KUKA KRL program: MyProgram_218().src

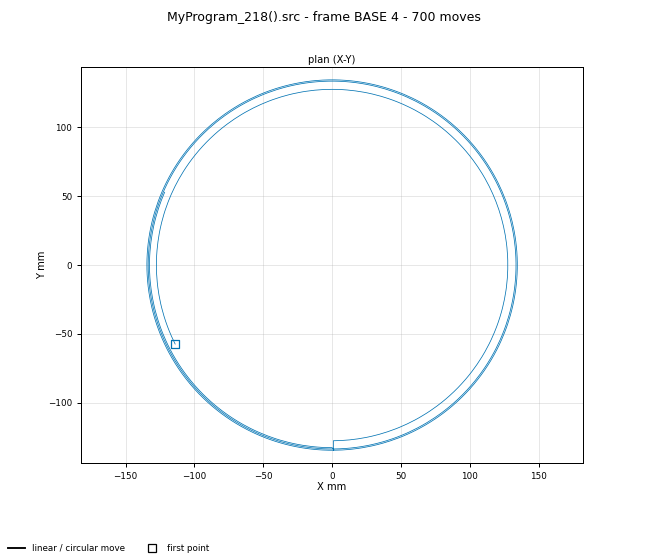
[picture p0: tool path of MyProgram_218().src in frame BASE 4, 700 of 700 moves have a stored position in this frame; points joined in program order, loops and branches not executed]
&ACCESS RVP
&REL 1
&PARAM TEMPLATE = C:\KRC\Roboter\Template\vorgabe
&PARAM EDITMASK = *
DEF MyProgram_218()
; ---- Setting reference (Base) ----
$BASE = BASE_DATA[4]

; --------------------------
; ---- Setting tool (TCP) ----
$TOOL = TOOL_DATA[3]
; --------------------------

$VEL.CP = VEL_APROX_PRINT
Startdeposition()
$VEL.CP = VEL_PRINT
LIN {X -113.9727,Y -57.3713,Z 152,A -154.6859,B 17.5235,C -0.3256,E1 17.383,E2 243.3579} C_DIS
LIN {X -115.3507,Y -54.5472,Z 152,A -156.1373,B 17.5235,C -0.3282,E1 17.3813,E2 244.8124} C_DIS
LIN {X -116.579,Y -51.8684,Z 152,A -157.511,B 17.5234,C -0.3302,E1 17.3797,E2 246.1904} C_DIS
LIN {X -118.2068,Y -48.044,Z 152,A -159.4681,B 17.5234,C -0.3326,E1 17.3776,E2 248.1558} C_DIS
LIN {X -119.5357,Y -44.6339,Z 152,A -161.0343,B 17.5232,C -0.3396,E1 17.376,E2 249.7114} C_DIS
LIN {X -120.8839,Y -40.8453,Z 152,A -162.9985,B 17.5232,C -0.3398,E1 17.3742,E2 251.6915} C_DIS
LIN {X -122.0836,Y -37.1027,Z 152,A -164.6161,B 17.523,C -0.3495,E1 17.3729,E2 253.2904} C_DIS
LIN {X -122.9269,Y -34.2049,Z 152,A -165.9736,B 17.523,C -0.3534,E1 17.3718,E2 254.6466} C_DIS
LIN {X -123.7291,Y -31.1788,Z 152,A -167.3908,B 17.5229,C -0.3571,E1 17.3708,E2 256.0634} C_DIS
LIN {X -124.4565,Y -28.1362,Z 152,A -168.7811,B 17.5228,C -0.3617,E1 17.37,E2 257.4504} C_DIS
LIN {X -125.1457,Y -24.8967,Z 152,A -170.2929,B 17.5227,C -0.3654,E1 17.3691,E2 258.9631} C_DIS
LIN {X -125.7207,Y -21.8119,Z 152,A -171.7167,B 17.5227,C -0.3691,E1 17.3684,E2 260.3869} C_DIS
LIN {X -126.2175,Y -18.7245,Z 152,A -173.1623,B 17.5226,C -0.3721,E1 17.3678,E2 261.8354} C_DIS
LIN {X -126.5469,Y -16.3393,Z 152,A -174.3275,B 17.5226,C -0.3728,E1 17.3674,E2 263.0086} C_DIS
LIN {X -126.9668,Y -12.6766,Z 152,A -175.922,B 17.5224,C -0.3797,E1 17.3669,E2 264.5941} C_DIS
LIN {X -127.2461,Y -9.4608,Z 152,A -177.3928,B 17.5224,C -0.3834,E1 17.3666,E2 266.0654} C_DIS
LIN {X -127.4345,Y -6.4427,Z 152,A -178.7722,B 17.5222,C -0.3869,E1 17.3663,E2 267.4454} C_DIS
LIN {X -127.5543,Y -3.3188,Z 152,A 179.8307,B 17.5222,C -0.3914,E1 17.3663,E2 268.8398} C_DIS
LIN {X -127.6001,Y -0.0843,Z 152,A 178.3637,B 17.5221,C -0.3954,E1 17.3662,E2 270.3066} C_DIS
LIN {X -127.5647,Y 2.9425,Z 152,A 176.9278,B 17.5221,C -0.3972,E1 17.3662,E2 271.7492} C_DIS
LIN {X -127.4125,Y 6.8803,Z 152,A 175.04,B 17.522,C -0.399,E1 17.3665,E2 273.6477} C_DIS
LIN {X -127.1428,Y 10.7584,Z 152,A 173.4238,B 17.5218,C -0.4084,E1 17.3668,E2 275.247} C_DIS
LIN {X -126.8198,Y 14.0691,Z 152,A 171.9562,B 17.5217,C -0.4138,E1 17.3673,E2 276.7095} C_DIS
LIN {X -126.4609,Y 16.9953,Z 152,A 170.6184,B 17.5216,C -0.4174,E1 17.3677,E2 278.0471} C_DIS
LIN {X -126.007,Y 20.0892,Z 152,A 169.1704,B 17.5216,C -0.4203,E1 17.3684,E2 279.498} C_DIS
LIN {X -125.4777,Y 23.1701,Z 152,A 167.7181,B 17.5214,C -0.4231,E1 17.3691,E2 280.9538} C_DIS
LIN {X -124.7928,Y 26.6056,Z 152,A 166.0587,B 17.5214,C -0.4252,E1 17.37,E2 282.6206} C_DIS
LIN {X -123.7662,Y 31.0327,Z 152,A 164.1264,B 17.5212,C -0.4347,E1 17.3713,E2 284.5378} C_DIS
LIN {X -122.9699,Y 34.0512,Z 152,A 162.8468,B 17.521,C -0.4427,E1 17.3722,E2 285.8017} C_DIS
LIN {X -122.1521,Y 36.8791,Z 152,A 161.3808,B 17.521,C -0.4422,E1 17.3733,E2 287.2819} C_DIS
LIN {X -121.2101,Y 39.8659,Z 152,A 159.9672,B 17.5209,C -0.4461,E1 17.3745,E2 288.6944} C_DIS
LIN {X -120.1418,Y 42.9767,Z 152,A 158.4732,B 17.5208,C -0.4499,E1 17.3759,E2 290.1881} C_DIS
LIN {X -119.0471,Y 45.9221,Z 152,A 157.0498,B 17.5207,C -0.4537,E1 17.3773,E2 291.6109} C_DIS
LIN {X -118.0113,Y 48.5257,Z 152,A 155.7284,B 17.5207,C -0.4553,E1 17.3787,E2 292.9376} C_DIS
LIN {X -116.8398,Y 51.2823,Z 152,A 154.2995,B 17.5207,C -0.4566,E1 17.3803,E2 294.3739} C_DIS
LIN {X -115.4259,Y 54.3898,Z 152,A 152.885,B 17.5204,C -0.4646,E1 17.382,E2 295.773} C_DIS
LIN {X -114.0589,Y 57.202,Z 152,A 151.456,B 17.5204,C -0.4678,E1 17.3837,E2 297.2028} C_DIS
LIN {X -112.5261,Y 60.1611,Z 152,A 149.9928,B 17.5202,C -0.473,E1 17.3856,E2 298.6602} C_DIS
LIN {X -111.11,Y 62.7379,Z 152,A 148.593,B 17.5202,C -0.4741,E1 17.3875,E2 300.0669} C_DIS
LIN {X -109.5435,Y 65.4343,Z 152,A 147.208,B 17.5201,C -0.4784,E1 17.3895,E2 301.4483} C_DIS
LIN {X -107.9124,Y 68.0906,Z 152,A 145.7625,B 17.52,C -0.4807,E1 17.3916,E2 302.8969} C_DIS
LIN {X -106.0955,Y 70.8884,Z 152,A 144.2532,B 17.52,C -0.4843,E1 17.3939,E2 304.4053} C_DIS
LIN {X -103.8442,Y 74.1471,Z 152,A 142.3482,B 17.5199,C -0.485,E1 17.397,E2 306.322} C_DIS
LIN {X -101.547,Y 77.264,Z 152,A 140.7503,B 17.5196,C -0.4938,E1 17.3997,E2 307.9018} C_DIS
LIN {X -99.1877,Y 80.2699,Z 152,A 139.0108,B 17.5196,C -0.4973,E1 17.4027,E2 309.6417} C_DIS
LIN {X -96.9265,Y 82.9868,Z 152,A 137.3158,B 17.5196,C -0.4978,E1 17.4058,E2 311.3465} C_DIS
LIN {X -94.0753,Y 86.2049,Z 152,A 135.4528,B 17.5193,C -0.5045,E1 17.4092,E2 313.1994} C_DIS
LIN {X -91.3904,Y 89.047,Z 152,A 133.6596,B 17.5193,C -0.5073,E1 17.4127,E2 314.9945} C_DIS
LIN {X -88.5541,Y 91.8676,Z 152,A 131.745,B 17.5193,C -0.5076,E1 17.4165,E2 316.9199} C_DIS
LIN {X -85.3855,Y 94.82,Z 152,A 129.8494,B 17.5191,C -0.5134,E1 17.4204,E2 318.8076} C_DIS
LIN {X -82.6808,Y 97.1869,Z 152,A 128.179,B 17.5191,C -0.515,E1 17.4239,E2 320.4823} C_DIS
LIN {X -79.7356,Y 99.6181,Z 152,A 126.4292,B 17.519,C -0.5174,E1 17.4277,E2 322.2338} C_DIS
LIN {X -76.1604,Y 102.3768,Z 152,A 124.5451,B 17.5187,C -0.5259,E1 17.4319,E2 324.0995} C_DIS
LIN {X -73.4698,Y 104.3245,Z 152,A 123.0566,B 17.5187,C -0.5288,E1 17.4353,E2 325.586} C_DIS
LIN {X -70.9621,Y 106.0463,Z 152,A 121.6854,B 17.5186,C -0.5311,E1 17.4384,E2 326.9561} C_DIS
LIN {X -68.3819,Y 107.7285,Z 152,A 120.2468,B 17.5186,C -0.5318,E1 17.4418,E2 328.3994} C_DIS
LIN {X -66.0845,Y 109.1524,Z 152,A 118.9664,B 17.5186,C -0.5318,E1 17.4449,E2 329.6858} C_DIS
LIN {X -63.0785,Y 110.9168,Z 152,A 117.4551,B 17.5184,C -0.536,E1 17.4485,E2 331.1894} C_DIS
LIN {X -60.1402,Y 112.5374,Z 152,A 115.9589,B 17.5184,C -0.5387,E1 17.4522,E2 332.6828} C_DIS
LIN {X -57.3655,Y 113.9757,Z 152,A 114.5616,B 17.5183,C -0.541,E1 17.4557,E2 334.0779} C_DIS
LIN {X -54.5551,Y 115.3469,Z 152,A 113.1534,B 17.5183,C -0.5429,E1 17.4592,E2 335.4852} C_DIS
LIN {X -51.8611,Y 116.5822,Z 152,A 111.7973,B 17.5183,C -0.544,E1 17.4627,E2 336.8427} C_DIS
LIN {X -48.8285,Y 117.8849,Z 152,A 110.3545,B 17.5181,C -0.5472,E1 17.4664,E2 338.2797} C_DIS
LIN {X -46.0972,Y 118.979,Z 152,A 109.0078,B 17.5181,C -0.548,E1 17.4699,E2 339.628} C_DIS
LIN {X -43.1738,Y 120.0707,Z 152,A 107.6953,B 17.5179,C -0.5525,E1 17.4733,E2 340.9292} C_DIS
LIN {X -40.016,Y 121.1601,Z 152,A 106.1214,B 17.5179,C -0.5517,E1 17.4774,E2 342.5101} C_DIS
LIN {X -37.0357,Y 122.1041,Z 152,A 104.6891,B 17.5179,C -0.5523,E1 17.4813,E2 343.9443} C_DIS
LIN {X -34.2041,Y 122.9271,Z 152,A 103.3614,B 17.5179,C -0.5534,E1 17.4848,E2 345.2714} C_DIS
LIN {X -31.1786,Y 123.7292,Z 152,A 101.9534,B 17.5179,C -0.5546,E1 17.4886,E2 346.6785} C_DIS
LIN {X -28.1119,Y 124.462,Z 152,A 100.5355,B 17.5179,C -0.5556,E1 17.4925,E2 348.0956} C_DIS
LIN {X -24.8793,Y 125.1493,Z 152,A 99.0624,B 17.5179,C -0.5571,E1 17.4965,E2 349.5664} C_DIS
LIN {X -21.8085,Y 125.7213,Z 152,A 97.6548,B 17.5178,C -0.5578,E1 17.5004,E2 350.9735} C_DIS
LIN {X -19.1709,Y 126.1492,Z 152,A 96.324,B 17.5178,C -0.5542,E1 17.5041,E2 352.3181} C_DIS
LIN {X -15.5304,Y 126.6491,Z 152,A 94.8319,B 17.5178,C -0.5603,E1 17.5082,E2 353.7915} C_DIS
LIN {X -12.6253,Y 126.9717,Z 152,A 93.4661,B 17.5178,C -0.5591,E1 17.512,E2 355.1625} C_DIS
LIN {X -9.3696,Y 127.2527,Z 152,A 92.0232,B 17.5178,C -0.5605,E1 17.516,E2 356.6018} C_DIS
LIN {X -6.6201,Y 127.4255,Z 152,A 90.6884,B 17.5178,C -0.5576,E1 17.5197,E2 357.9468} C_DIS
LIN {X -3.2848,Y 127.5552,Z 152,A 89.2597,B 17.5178,C -0.5603,E1 17.5237,E2 359.3668} C_DIS
LIN {X -0.2372,Y 127.5979,Z 152,A 87.8455,B 17.5178,C -0.5589,E1 17.5277,E2 360.7856} C_DIS
LIN {X 3.1496,Y 127.559,Z 152,A 86.198,B 17.5178,C -0.5547,E1 17.5323,E2 362.4465} C_DIS
LIN {X 7.5474,Y 127.3741,Z 152,A 84.3585,B 17.5178,C -0.5593,E1 17.5374,E2 364.2698} C_DIS
LIN {X 10.7934,Y 127.1398,Z 152,A 82.9113,B 17.5178,C -0.5596,E1 17.5414,E2 365.7148} C_DIS
LIN {X 14.0805,Y 126.8186,Z 152,A 81.4639,B 17.5177,C -0.5605,E1 17.5454,E2 367.1578} C_DIS
LIN {X 17.0025,Y 126.4599,Z 152,A 80.1413,B 17.5177,C -0.5602,E1 17.5491,E2 368.4801} C_DIS
LIN {X 20.0911,Y 126.0067,Z 152,A 78.7462,B 17.5177,C -0.5599,E1 17.5529,E2 369.8741} C_DIS
LIN {X 23.1858,Y 125.4748,Z 152,A 77.2629,B 17.5178,C -0.5568,E1 17.557,E2 371.3652} C_DIS
LIN {X 26.1682,Y 124.887,Z 152,A 75.8682,B 17.5178,C -0.5551,E1 17.5609,E2 372.7631} C_DIS
LIN {X 29.3622,Y 124.1739,Z 152,A 74.4493,B 17.5178,C -0.556,E1 17.5647,E2 374.176} C_DIS
LIN {X 32.5203,Y 123.3837,Z 152,A 73.0323,B 17.5178,C -0.5566,E1 17.5685,E2 375.5877} C_DIS
LIN {X 35.5353,Y 122.5492,Z 152,A 71.7806,B 17.5177,C -0.5609,E1 17.5718,E2 376.822} C_DIS
LIN {X 38.3685,Y 121.6924,Z 152,A 70.3268,B 17.5179,C -0.5555,E1 17.5758,E2 378.2899} C_DIS
LIN {X 40.7446,Y 120.9175,Z 152,A 69.0061,B 17.5181,C -0.5476,E1 17.5793,E2 379.6329} C_DIS
LIN {X 44.4806,Y 119.5931,Z 152,A 67.4143,B 17.5179,C -0.5526,E1 17.5834,E2 381.2035} C_DIS
LIN {X 47.5572,Y 118.403,Z 152,A 65.8169,B 17.5181,C -0.547,E1 17.5876,E2 382.814} C_DIS
LIN {X 51.5368,Y 116.7273,Z 152,A 63.9492,B 17.5181,C -0.5473,E1 17.5924,E2 384.674} C_DIS
LIN {X 54.395,Y 115.4234,Z 152,A 62.6043,B 17.5181,C -0.548,E1 17.5958,E2 386.0116} C_DIS
LIN {X 56.6861,Y 114.3139,Z 152,A 61.3941,B 17.5181,C -0.5442,E1 17.5988,E2 387.2295} C_DIS
LIN {X 60.1523,Y 112.5309,Z 152,A 59.7483,B 17.5181,C -0.5456,E1 17.6029,E2 388.8639} C_DIS
LIN {X 62.7654,Y 111.0945,Z 152,A 58.3557,B 17.5183,C -0.5418,E1 17.6063,E2 390.263} C_DIS
LIN {X 65.229,Y 109.6659,Z 152,A 57.0551,B 17.5183,C -0.5392,E1 17.6094,E2 391.5664} C_DIS
LIN {X 68.0911,Y 107.9121,Z 152,A 55.569,B 17.5183,C -0.5377,E1 17.6129,E2 393.0505} C_DIS
LIN {X 70.8752,Y 106.1043,Z 152,A 54.1195,B 17.5184,C -0.5368,E1 17.6163,E2 394.4959} C_DIS
LIN {X 73.4692,Y 104.3249,Z 152,A 52.6793,B 17.5185,C -0.5335,E1 17.6196,E2 395.9398} C_DIS
LIN {X 76.6358,Y 102.0218,Z 152,A 50.8146,B 17.5187,C -0.5266,E1 17.6238,E2 397.8173} C_DIS
LIN {X 80.2759,Y 99.1829,Z 152,A 48.9031,B 17.5187,C -0.5287,E1 17.628,E2 399.7115} C_DIS
LIN {X 82.8559,Y 97.038,Z 152,A 47.2561,B 17.5189,C -0.5208,E1 17.6315,E2 401.3752} C_DIS
LIN {X 86.2638,Y 94.0212,Z 152,A 45.2244,B 17.5189,C -0.5172,E1 17.6358,E2 403.4065} C_DIS
LIN {X 89.5956,Y 90.8524,Z 152,A 43.4329,B 17.5189,C -0.5229,E1 17.6393,E2 405.1683} C_DIS
LIN {X 91.8787,Y 88.5426,Z 152,A 41.7138,B 17.5192,C -0.5103,E1 17.6427,E2 406.918} C_DIS
LIN {X 95.0101,Y 85.1734,Z 152,A 39.8051,B 17.5192,C -0.5115,E1 17.6463,E2 408.8103} C_DIS
LIN {X 97.1851,Y 82.6829,Z 152,A 38.2159,B 17.5194,C -0.5044,E1 17.6492,E2 410.4124} C_DIS
LIN {X 99.6158,Y 79.7385,Z 152,A 36.4998,B 17.5194,C -0.5004,E1 17.6522,E2 412.13} C_DIS
LIN {X 102.2461,Y 76.3359,Z 152,A 34.81,B 17.5194,C -0.5047,E1 17.655,E2 413.7938} C_DIS
LIN {X 104.2367,Y 73.5943,Z 152,A 33.2206,B 17.5195,C -0.4985,E1 17.6576,E2 415.3923} C_DIS
LIN {X 105.7394,Y 71.4185,Z 152,A 31.9523,B 17.5197,C -0.4926,E1 17.6596,E2 416.6707} C_DIS
LIN {X 107.7055,Y 68.4184,Z 152,A 30.3969,B 17.5197,C -0.4906,E1 17.662,E2 418.2213} C_DIS
LIN {X 109.1695,Y 66.0563,Z 152,A 29.1069,B 17.5199,C -0.4858,E1 17.6639,E2 419.5172} C_DIS
LIN {X 110.9329,Y 63.0503,Z 152,A 27.6196,B 17.5199,C -0.4846,E1 17.6659,E2 420.9971} C_DIS
LIN {X 112.5301,Y 60.1537,Z 152,A 26.1549,B 17.5199,C -0.4815,E1 17.6679,E2 422.4609} C_DIS
LIN {X 113.974,Y 57.3689,Z 152,A 24.7695,B 17.5201,C -0.4786,E1 17.6697,E2 423.845} C_DIS
LIN {X 115.3525,Y 54.5434,Z 152,A 23.4063,B 17.5201,C -0.4765,E1 17.6713,E2 425.2042} C_DIS
LIN {X 116.5781,Y 51.8704,Z 152,A 22.0428,B 17.5202,C -0.4713,E1 17.6729,E2 426.574} C_DIS
LIN {X 117.8808,Y 48.8383,Z 152,A 20.6189,B 17.5202,C -0.4694,E1 17.6744,E2 427.9928} C_DIS
LIN {X 118.9736,Y 46.111,Z 152,A 19.2844,B 17.5204,C -0.4651,E1 17.6758,E2 429.3304} C_DIS
LIN {X 120.0763,Y 43.1585,Z 152,A 17.8852,B 17.5204,C -0.4617,E1 17.6771,E2 430.7294} C_DIS
LIN {X 121.0836,Y 40.2459,Z 152,A 16.5038,B 17.5206,C -0.4578,E1 17.6784,E2 432.112} C_DIS
LIN {X 122.1039,Y 37.0365,Z 152,A 15.0152,B 17.5206,C -0.4543,E1 17.6796,E2 433.5998} C_DIS
LIN {X 122.9263,Y 34.2069,Z 152,A 13.7032,B 17.5208,C -0.4509,E1 17.6806,E2 434.9119} C_DIS
LIN {X 123.728,Y 31.1835,Z 152,A 12.3118,B 17.5208,C -0.4472,E1 17.6816,E2 436.3035} C_DIS
LIN {X 124.4575,Y 28.1319,Z 152,A 10.917,B 17.5209,C -0.4436,E1 17.6825,E2 437.6985} C_DIS
LIN {X 125.1485,Y 24.883,Z 152,A 9.4528,B 17.521,C -0.4401,E1 17.6833,E2 439.1614} C_DIS
LIN {X 125.7205,Y 21.8133,Z 152,A 8.0609,B 17.5211,C -0.4363,E1 17.684,E2 440.5539} C_DIS
LIN {X 126.2166,Y 18.7312,Z 152,A 6.6205,B 17.5213,C -0.4306,E1 17.6846,E2 442.0005} C_DIS
LIN {X 126.6434,Y 15.5787,Z 152,A 5.2902,B 17.5213,C -0.43,E1 17.6851,E2 443.3214} C_DIS
LIN {X 126.9682,Y 12.6619,Z 152,A 3.9262,B 17.5214,C -0.4243,E1 17.6855,E2 444.6924} C_DIS
LIN {X 127.2517,Y 9.3841,Z 152,A 2.4704,B 17.5214,C -0.4206,E1 17.6858,E2 446.1476} C_DIS
LIN {X 127.4339,Y 6.4536,Z 152,A 1.1297,B 17.5216,C -0.4157,E1 17.686,E2 447.4926} C_DIS
LIN {X 127.5549,Y 3.2971,Z 152,A -0.2217,B 17.5216,C -0.4139,E1 17.6861,E2 448.8383} C_DIS
LIN {X 127.5999,Y -0.1226,Z 152,A -1.735,B 17.5217,C -0.4099,E1 17.6861,E2 450.3511} C_DIS
LIN {X 127.5635,Y -2.9879,Z 152,A -3.0967,B 17.5219,C -0.4032,E1 17.6861,E2 451.7232} C_DIS
LIN {X 127.4535,Y -6.0634,Z 152,A -4.4675,B 17.5219,C -0.3994,E1 17.6859,E2 453.0946} C_DIS
LIN {X 127.2627,Y -9.2329,Z 152,A -5.8219,B 17.522,C -0.3977,E1 17.6857,E2 454.4427} C_DIS
LIN {X 126.9816,Y -12.5221,Z 152,A -7.281,B 17.522,C -0.394,E1 17.6853,E2 455.9013} C_DIS
LIN {X 126.6378,Y -15.6255,Z 152,A -8.6566,B 17.5222,C -0.3906,E1 17.6849,E2 457.2758} C_DIS
LIN {X 126.2438,Y -18.5407,Z 152,A -9.9788,B 17.5222,C -0.3866,E1 17.6844,E2 458.6} C_DIS
LIN {X 125.7181,Y -21.8264,Z 152,A -11.4215,B 17.5223,C -0.3839,E1 17.6837,E2 460.0389} C_DIS
LIN {X 125.1456,Y -24.8975,Z 152,A -12.8014,B 17.5223,C -0.3805,E1 17.683,E2 461.4182} C_DIS
LIN {X 124.497,Y -27.9587,Z 152,A -14.126,B 17.5224,C -0.3793,E1 17.6822,E2 462.7355} C_DIS
LIN {X 123.7741,Y -31.0017,Z 152,A -15.647,B 17.5226,C -0.3706,E1 17.6812,E2 464.2721} C_DIS
LIN {X 122.9768,Y -34.0263,Z 152,A -17.0374,B 17.5226,C -0.3669,E1 17.6802,E2 465.6628} C_DIS
LIN {X 121.9537,Y -37.5271,Z 152,A -18.6757,B 17.5228,C -0.362,E1 17.6789,E2 467.3036} C_DIS
LIN {X 120.7154,Y -41.3398,Z 152,A -20.5043,B 17.5228,C -0.3556,E1 17.6773,E2 469.1381} C_DIS
LIN {X 119.5324,Y -44.6426,Z 152,A -22.1216,B 17.523,C -0.3494,E1 17.6757,E2 470.7624} C_DIS
LIN {X 117.8814,Y -48.8368,Z 152,A -23.9488,B 17.523,C -0.3509,E1 17.6738,E2 472.5699} C_DIS
LIN {X 116.7231,Y -51.5461,Z 152,A -25.3771,B 17.5231,C -0.3431,E1 17.6722,E2 474.0123} C_DIS
LIN {X 115.4269,Y -54.3877,Z 152,A -26.7063,B 17.5231,C -0.3418,E1 17.6707,E2 475.335} C_DIS
LIN {X 114.0623,Y -57.1954,Z 152,A -28.1026,B 17.5232,C -0.3381,E1 17.6689,E2 476.7327} C_DIS
LIN {X 112.5434,Y -60.1289,Z 152,A -29.5443,B 17.5232,C -0.3355,E1 17.6671,E2 478.1718} C_DIS
LIN {X 111.0232,Y -62.8921,Z 152,A -31.1308,B 17.5235,C -0.3252,E1 17.6649,E2 479.7801} C_DIS
LIN {X 108.7235,Y -66.7878,Z 152,A -32.9962,B 17.5235,C -0.3259,E1 17.6622,E2 481.6291} C_DIS
LIN {X 106.9561,Y -69.5831,Z 152,A -34.4704,B 17.5235,C -0.3223,E1 17.66,E2 483.1041} C_DIS
LIN {X 105.2184,Y -72.1837,Z 152,A -35.8035,B 17.5235,C -0.3213,E1 17.6579,E2 484.4309} C_DIS
LIN {X 103.4052,Y -74.7583,Z 152,A -37.2614,B 17.5236,C -0.3159,E1 17.6555,E2 485.8959} C_DIS
LIN {X 101.5429,Y -77.2693,Z 152,A -38.6513,B 17.5236,C -0.3129,E1 17.6532,E2 487.2861} C_DIS
LIN {X 99.1856,Y -80.2724,Z 152,A -40.3639,B 17.5238,C -0.3086,E1 17.6502,E2 489.001} C_DIS
LIN {X 97.0943,Y -82.7898,Z 152,A -41.9717,B 17.5238,C -0.2999,E1 17.6473,E2 490.6267} C_DIS
LIN {X 94.0701,Y -86.2105,Z 152,A -43.8726,B 17.5238,C -0.3005,E1 17.6438,E2 492.5131} C_DIS
LIN {X 91.3874,Y -89.0501,Z 152,A -45.6394,B 17.524,C -0.2959,E1 17.6404,E2 494.2838} C_DIS
LIN {X 88.5537,Y -91.868,Z 152,A -47.5442,B 17.524,C -0.2878,E1 17.6365,E2 496.2036} C_DIS
LIN {X 85.1685,Y -95.0144,Z 152,A -49.459,B 17.524,C -0.2891,E1 17.6326,E2 498.1025} C_DIS
LIN {X 82.6786,Y -97.1888,Z 152,A -51.0484,B 17.5242,C -0.2821,E1 17.6292,E2 499.706} C_DIS
LIN {X 79.7344,Y -99.6191,Z 152,A -52.7656,B 17.5242,C -0.2784,E1 17.6255,E2 501.4257} C_DIS
LIN {X 76.1486,Y -102.3856,Z 152,A -54.6422,B 17.5242,C -0.2801,E1 17.6214,E2 503.2866} C_DIS
LIN {X 73.6188,Y -104.2195,Z 152,A -56.0343,B 17.5242,C -0.2778,E1 17.6182,E2 504.6791} C_DIS
LIN {X 71.0407,Y -105.9938,Z 152,A -57.4285,B 17.5242,C -0.2756,E1 17.615,E2 506.0736} C_DIS
LIN {X 68.4247,Y -107.7015,Z 152,A -58.8742,B 17.5243,C -0.2715,E1 17.6116,E2 507.5259} C_DIS
LIN {X 65.6278,Y -109.4282,Z 152,A -60.3035,B 17.5243,C -0.2706,E1 17.6082,E2 508.9514} C_DIS
LIN {X 63.4871,Y -110.6837,Z 152,A -61.5477,B 17.5245,C -0.264,E1 17.6051,E2 510.212} C_DIS
LIN {X 60.1265,Y -112.5447,Z 152,A -63.1414,B 17.5245,C -0.266,E1 17.6013,E2 511.7923} C_DIS
LIN {X 57.3554,Y -113.9808,Z 152,A -64.5249,B 17.5245,C -0.2645,E1 17.5978,E2 513.1752} C_DIS
LIN {X 54.5498,Y -115.3494,Z 152,A -65.9184,B 17.5245,C -0.2627,E1 17.5943,E2 514.5692} C_DIS
LIN {X 51.8741,Y -116.5764,Z 152,A -67.255,B 17.5245,C -0.2603,E1 17.5909,E2 515.9088} C_DIS
LIN {X 48.8391,Y -117.8805,Z 152,A -68.6861,B 17.5245,C -0.2602,E1 17.5872,E2 517.3354} C_DIS
LIN {X 46.4601,Y -118.838,Z 152,A -69.9394,B 17.5245,C -0.255,E1 17.5839,E2 518.6015} C_DIS
LIN {X 43.1564,Y -120.077,Z 152,A -71.4338,B 17.5245,C -0.2563,E1 17.58,E2 520.0869} C_DIS
LIN {X 40.2404,Y -121.0854,Z 152,A -72.8222,B 17.5245,C -0.2546,E1 17.5764,E2 521.477} C_DIS
LIN {X 37.0295,Y -122.106,Z 152,A -74.2684,B 17.5245,C -0.2554,E1 17.5725,E2 522.9167} C_DIS
LIN {X 34.1969,Y -122.9291,Z 152,A -75.6414,B 17.5246,C -0.2523,E1 17.5688,E2 524.2966} C_DIS
LIN {X 31.1748,Y -123.7302,Z 152,A -77.0405,B 17.5246,C -0.2512,E1 17.565,E2 525.6963} C_DIS
LIN {X 28.5399,Y -124.3643,Z 152,A -78.3409,B 17.5246,C -0.2472,E1 17.5615,E2 527.0072} C_DIS
LIN {X 24.837,Y -125.1579,Z 152,A -79.9367,B 17.5246,C -0.2495,E1 17.5571,E2 528.5923} C_DIS
LIN {X 21.7826,Y -125.726,Z 152,A -81.3305,B 17.5246,C -0.2485,E1 17.5533,E2 529.987} C_DIS
LIN {X 18.7118,Y -126.2194,Z 152,A -82.7491,B 17.5246,C -0.2469,E1 17.5494,E2 531.4091} C_DIS
LIN {X 15.6262,Y -126.6377,Z 152,A -84.0807,B 17.5246,C -0.2484,E1 17.5457,E2 532.7339} C_DIS
LIN {X 12.7136,Y -126.9633,Z 152,A -85.4586,B 17.5247,C -0.2456,E1 17.5419,E2 534.1198} C_DIS
LIN {X 9.4289,Y -127.2484,Z 152,A -86.9003,B 17.5247,C -0.2463,E1 17.5379,E2 535.5579} C_DIS
LIN {X 6.4429,Y -127.4345,Z 152,A -88.2979,B 17.5247,C -0.244,E1 17.534,E2 536.9625} C_DIS
LIN {X 3.684,Y -127.5441,Z 152,A -89.5932,B 17.5247,C -0.2417,E1 17.5303,E2 538.2648} C_DIS
LIN {X 0.9105,Y -127.5933,Z 152,A -90.4609,B 17.5246,C -0.2546,E1 17.528,E2 539.0895} C_DIS
Enddeposition()
LIN {X 0.9478,Y -134.4897,Z 153,A -92.8925,B 24.9696,C -1.2741,E1 25.0007,E2 539.514} C_DIS
Startdeposition()
$VEL.CP = VEL_PRINT
LIN {X -2.5634,Y -134.4703,Z 153,A -94.5447,B 24.97,C -1.2655,E1 24.996,E2 541.1866} C_DIS
LIN {X -6.9086,Y -134.3168,Z 153,A -96.3362,B 24.9699,C -1.2685,E1 24.991,E2 542.9712} C_DIS
LIN {X -10.8072,Y -134.0603,Z 153,A -98.0755,B 24.97,C -1.2646,E1 24.9861,E2 544.7206} C_DIS
LIN {X -15.072,Y -133.6488,Z 153,A -99.9353,B 24.9701,C -1.263,E1 24.981,E2 546.5853} C_DIS
LIN {X -19.01,Y -133.1439,Z 153,A -101.5224,B 24.9698,C -1.2688,E1 24.9766,E2 548.1598} C_DIS
LIN {X -22.9533,Y -132.5231,Z 153,A -103.3167,B 24.9701,C -1.2644,E1 24.9716,E2 549.9662} C_DIS
LIN {X -26.8096,Y -131.7949,Z 153,A -104.8838,B 24.9698,C -1.2706,E1 24.9674,E2 551.5204} C_DIS
LIN {X -30.0715,Y -131.0891,Z 153,A -106.3278,B 24.9698,C -1.2702,E1 24.9634,E2 552.9673} C_DIS
LIN {X -33.8277,Y -130.1726,Z 153,A -108.0979,B 24.97,C -1.2647,E1 24.9586,E2 554.7528} C_DIS
LIN {X -37.6662,Y -129.112,Z 153,A -109.6486,B 24.9696,C -1.2734,E1 24.9545,E2 556.2853} C_DIS
LIN {X -41.1809,Y -128.0344,Z 153,A -111.2459,B 24.9696,C -1.273,E1 24.9502,E2 557.8863} C_DIS
LIN {X -44.7701,Y -126.8259,Z 153,A -113.1757,B 24.9704,C -1.2581,E1 24.945,E2 559.8553} C_DIS
LIN {X -48.0717,Y -125.6113,Z 153,A -114.2734,B 24.9693,C -1.2802,E1 24.9423,E2 560.903} C_DIS
LIN {X -52.007,Y -124.0318,Z 153,A -116.1547,B 24.9694,C -1.2782,E1 24.9374,E2 562.7931} C_DIS
LIN {X -55.4404,Y -122.5368,Z 153,A -117.7216,B 24.9692,C -1.2815,E1 24.9334,E2 564.356} C_DIS
LIN {X -58.3958,Y -121.1558,Z 153,A -119.1516,B 24.9692,C -1.2811,E1 24.9298,E2 565.7906} C_DIS
LIN {X -62.1856,Y -119.2546,Z 153,A -120.9818,B 24.9692,C -1.2822,E1 24.9252,E2 567.6231} C_DIS
LIN {X -66.0185,Y -117.178,Z 153,A -122.8544,B 24.9692,C -1.284,E1 24.9206,E2 569.4968} C_DIS
LIN {X -69.6616,Y -115.0494,Z 153,A -124.7164,B 24.9692,C -1.2834,E1 24.9162,E2 571.3659} C_DIS
LIN {X -73.231,Y -112.811,Z 153,A -126.5092,B 24.969,C -1.2863,E1 24.9119,E2 573.1574} C_DIS
LIN {X -77.0791,Y -110.218,Z 153,A -128.476,B 24.9688,C -1.2902,E1 24.9074,E2 575.1218} C_DIS
LIN {X -80.6725,Y -107.6161,Z 153,A -130.4268,B 24.9688,C -1.2904,E1 24.903,E2 577.0788} C_DIS
LIN {X -84.2762,Y -104.8173,Z 153,A -132.3295,B 24.9685,C -1.2962,E1 24.8989,E2 578.9749} C_DIS
LIN {X -87.6638,Y -102.0009,Z 153,A -134.1117,B 24.9681,C -1.3046,E1 24.8951,E2 580.7439} C_DIS
LIN {X -90.3119,Y -99.6638,Z 153,A -135.6758,B 24.9681,C -1.3046,E1 24.8918,E2 582.314} C_DIS
LIN {X -93.3537,Y -96.8207,Z 153,A -137.5009,B 24.9681,C -1.3058,E1 24.8881,E2 584.1439} C_DIS
LIN {X -96.7474,Y -93.4295,Z 153,A -139.5871,B 24.9679,C -1.3082,E1 24.884,E2 586.2334} C_DIS
LIN {X -99.6808,Y -90.2931,Z 153,A -141.4175,B 24.9677,C -1.3124,E1 24.8806,E2 588.062} C_DIS
LIN {X -102.7106,Y -86.8318,Z 153,A -143.108,B 24.9668,C -1.3304,E1 24.8775,E2 589.7173} C_DIS
LIN {X -105.9126,Y -82.8956,Z 153,A -145.6917,B 24.9676,C -1.3147,E1 24.8729,E2 592.3504} C_DIS
LIN {X -108.945,Y -78.8676,Z 153,A -147.6997,B 24.967,C -1.327,E1 24.8696,E2 594.3387} C_DIS
LIN {X -111.3761,Y -75.3954,Z 153,A -149.5306,B 24.9668,C -1.3305,E1 24.8667,E2 596.1705} C_DIS
LIN {X -113.9315,Y -71.4763,Z 153,A -151.5412,B 24.9666,C -1.3349,E1 24.8637,E2 598.1807} C_DIS
LIN {X -116.2658,Y -67.6123,Z 153,A -153.3947,B 24.9662,C -1.3436,E1 24.8611,E2 600.023} C_DIS
LIN {X -118.2884,Y -64.0087,Z 153,A -155.2431,B 24.9662,C -1.3442,E1 24.8586,E2 601.8798} C_DIS
LIN {X -120.0751,Y -60.5869,Z 153,A -156.938,B 24.966,C -1.3464,E1 24.8564,E2 603.5785} C_DIS
LIN {X -121.9458,Y -56.7265,Z 153,A -159.0307,B 24.9664,C -1.3387,E1 24.8539,E2 605.7008} C_DIS
LIN {X -123.4895,Y -53.2816,Z 153,A -160.2273,B 24.9652,C -1.3636,E1 24.8526,E2 606.8448} C_DIS
LIN {X -124.7249,Y -50.3219,Z 153,A -161.6661,B 24.9652,C -1.3641,E1 24.8511,E2 608.2904} C_DIS
LIN {X -125.9596,Y -47.1464,Z 153,A -163.0957,B 24.9649,C -1.3695,E1 24.8497,E2 609.715} C_DIS
LIN {X -127.0935,Y -43.9985,Z 153,A -164.5377,B 24.9647,C -1.3731,E1 24.8483,E2 611.1569} C_DIS
LIN {X -128.1459,Y -40.8319,Z 153,A -165.9702,B 24.9645,C -1.3769,E1 24.8471,E2 612.5884} C_DIS
LIN {X -129.1177,Y -37.6468,Z 153,A -167.3506,B 24.9642,C -1.3832,E1 24.846,E2 613.9619} C_DIS
LIN {X -130.0293,Y -34.3672,Z 153,A -168.7956,B 24.9639,C -1.388,E1 24.8449,E2 615.4038} C_DIS
LIN {X -130.8403,Y -31.1385,Z 153,A -170.3828,B 24.9641,C -1.3842,E1 24.8439,E2 617.0093} C_DIS
LIN {X -132.0338,Y -25.6097,Z 153,A -172.9547,B 24.9641,C -1.384,E1 24.8424,E2 619.5969} C_DIS
LIN {X -132.9894,Y -20.069,Z 153,A -175.2326,B 24.9634,C -1.3974,E1 24.8414,E2 621.8563} C_DIS
LIN {X -133.5863,Y -15.6046,Z 153,A -177.1262,B 24.963,C -1.4049,E1 24.8407,E2 623.7435} C_DIS
LIN {X -134.0194,Y -11.2915,Z 153,A -178.9145,B 24.9626,C -1.4138,E1 24.8403,E2 625.5213} C_DIS
LIN {X -134.305,Y -7.1449,Z 153,A 179.2772,B 24.9623,C -1.4178,E1 24.84,E2 627.331} C_DIS
LIN {X -134.4476,Y -3.5485,Z 153,A 177.7281,B 24.9621,C -1.4221,E1 24.8398,E2 628.8792} C_DIS
LIN {X -134.4917,Y 0.7945,Z 153,A 175.9557,B 24.9616,C -1.432,E1 24.8398,E2 630.6387} C_DIS
LIN {X -134.4247,Y 4.3751,Z 153,A 174.2375,B 24.9618,C -1.4276,E1 24.8399,E2 632.3775} C_DIS
LIN {X -134.2317,Y 8.4009,Z 153,A 172.6945,B 24.9611,C -1.4418,E1 24.8402,E2 633.8961} C_DIS
LIN {X -133.9913,Y 11.624,Z 153,A 171.242,B 24.9611,C -1.4427,E1 24.8405,E2 635.3552} C_DIS
LIN {X -133.5576,Y 15.8448,Z 153,A 169.4494,B 24.9606,C -1.4494,E1 24.841,E2 637.1425} C_DIS
LIN {X -133.1308,Y 19.1019,Z 153,A 167.984,B 24.9606,C -1.4508,E1 24.8416,E2 638.6133} C_DIS
LIN {X -132.449,Y 23.3672,Z 153,A 166.1115,B 24.9603,C -1.4553,E1 24.8424,E2 640.4862} C_DIS
LIN {X -131.7208,Y 27.174,Z 153,A 164.3936,B 24.9603,C -1.4575,E1 24.8434,E2 642.2091} C_DIS
LIN {X -130.7918,Y 31.3396,Z 153,A 162.6373,B 24.9597,C -1.4664,E1 24.8445,E2 643.9544} C_DIS
LIN {X -129.8804,Y 34.9254,Z 153,A 160.7446,B 24.9603,C -1.4562,E1 24.8459,E2 645.8824} C_DIS
LIN {X -128.8847,Y 38.4425,Z 153,A 159.5767,B 24.959,C -1.4801,E1 24.8467,E2 647.0002} C_DIS
LIN {X -127.073,Y 44.0574,Z 153,A 157.3256,B 24.9578,C -1.5009,E1 24.8487,E2 649.2145} C_DIS
LIN {X -126.2056,Y 46.4896,Z 153,A 155.7789,B 24.9588,C -1.4826,E1 24.8502,E2 650.8136} C_DIS
LIN {X -124.7896,Y 50.1615,Z 153,A 154.2267,B 24.9582,C -1.494,E1 24.8517,E2 652.3475} C_DIS
LIN {X -123.235,Y 53.8704,Z 153,A 152.509,B 24.9579,C -1.4991,E1 24.8536,E2 654.0625} C_DIS
LIN {X -121.9227,Y 56.7764,Z 153,A 151.1499,B 24.9577,C -1.5032,E1 24.8552,E2 655.4191} C_DIS
LIN {X -120.4553,Y 59.8267,Z 153,A 149.625,B 24.9577,C -1.5036,E1 24.8571,E2 656.9513} C_DIS
LIN {X -118.333,Y 63.9256,Z 153,A 147.7222,B 24.9571,C -1.5126,E1 24.8595,E2 658.8428} C_DIS
LIN {X -116.927,Y 66.4623,Z 153,A 146.3958,B 24.9571,C -1.5119,E1 24.8614,E2 660.178} C_DIS
LIN {X -114.7904,Y 70.0881,Z 153,A 144.5939,B 24.9569,C -1.5167,E1 24.8639,E2 661.9776} C_DIS
LIN {X -112.6349,Y 73.5023,Z 153,A 142.7994,B 24.9569,C -1.518,E1 24.8666,E2 663.778} C_DIS
LIN {X -110.1276,Y 77.2085,Z 153,A 140.8686,B 24.9566,C -1.5222,E1 24.8697,E2 665.7084} C_DIS
LIN {X -107.5157,Y 80.8056,Z 153,A 138.9593,B 24.9563,C -1.5267,E1 24.8729,E2 667.6162} C_DIS
LIN {X -104.8115,Y 84.2833,Z 153,A 137.0809,B 24.956,C -1.5318,E1 24.8761,E2 669.4914} C_DIS
LIN {X -101.2315,Y 88.5511,Z 153,A 134.8688,B 24.9552,C -1.5459,E1 24.8801,E2 671.6799} C_DIS
LIN {X -98.3244,Y 91.7683,Z 153,A 132.7886,B 24.9556,C -1.5393,E1 24.884,E2 673.7852} C_DIS
LIN {X -95.6745,Y 94.5284,Z 153,A 131.2103,B 24.9552,C -1.5459,E1 24.8871,E2 675.3545} C_DIS
LIN {X -92.5367,Y 97.6021,Z 153,A 129.3799,B 24.9548,C -1.5524,E1 24.8908,E2 677.1769} C_DIS
LIN {X -89.4409,Y 100.4468,Z 153,A 127.3191,B 24.9554,C -1.5434,E1 24.8951,E2 679.2675} C_DIS
LIN {X -86.9486,Y 102.6113,Z 153,A 125.4478,B 24.9565,C -1.5239,E1 24.8992,E2 681.1924} C_DIS
LIN {X -82.5009,Y 106.2201,Z 153,A 124.0381,B 24.9532,C -1.58,E1 24.902,E2 682.4739} C_DIS
LIN {X -78.019,Y 109.5546,Z 153,A 121.3773,B 24.9538,C -1.571,E1 24.9081,E2 685.1655} C_DIS
LIN {X -74.8922,Y 111.7154,Z 153,A 119.6244,B 24.954,C -1.5676,E1 24.9121,E2 686.9323} C_DIS
LIN {X -71.2774,Y 114.0557,Z 153,A 117.7876,B 24.9538,C -1.571,E1 24.9165,E2 688.7668} C_DIS
LIN {X -67.6222,Y 116.2601,Z 153,A 115.9591,B 24.9536,C -1.5739,E1 24.9209,E2 690.594} C_DIS
LIN {X -63.7634,Y 118.4202,Z 153,A 114.1229,B 24.9532,C -1.5796,E1 24.9253,E2 692.4219} C_DIS
LIN {X -60.7895,Y 119.9719,Z 153,A 112.7538,B 24.9529,C -1.5851,E1 24.9287,E2 693.7818} C_DIS
LIN {X -57.7063,Y 121.4852,Z 153,A 111.3161,B 24.9527,C -1.5887,E1 24.9323,E2 695.2146} C_DIS
LIN {X -54.8799,Y 122.7876,Z 153,A 109.9194,B 24.9527,C -1.5872,E1 24.9359,E2 696.6183} C_DIS
LIN {X -51.6163,Y 124.195,Z 153,A 108.4589,B 24.9525,C -1.5921,E1 24.9396,E2 698.0705} C_DIS
LIN {X -48.5018,Y 125.4441,Z 153,A 106.987,B 24.9525,C -1.592,E1 24.9435,E2 699.5459} C_DIS
LIN {X -45.1209,Y 126.7004,Z 153,A 105.4031,B 24.9525,C -1.5916,E1 24.9476,E2 701.1339} C_DIS
LIN {X -41.269,Y 128.0063,Z 153,A 103.6872,B 24.9524,C -1.5946,E1 24.9522,E2 702.8459} C_DIS
LIN {X -37.8801,Y 129.0493,Z 153,A 102.1785,B 24.9522,C -1.5964,E1 24.9562,E2 704.3528} C_DIS
LIN {X -34.4479,Y 130.0078,Z 153,A 100.6999,B 24.952,C -1.6,E1 24.9602,E2 705.8252} C_DIS
LIN {X -30.9825,Y 130.8779,Z 153,A 99.1733,B 24.952,C -1.6012,E1 24.9643,E2 707.3509} C_DIS
LIN {X -26.9771,Y 131.7608,Z 153,A 97.4091,B 24.952,C -1.6019,E1 24.9691,E2 709.1156} C_DIS
LIN {X -23.3442,Y 132.4531,Z 153,A 95.8261,B 24.9519,C -1.6028,E1 24.9735,E2 710.6982} C_DIS
LIN {X -19.1714,Y 133.1208,Z 153,A 93.9745,B 24.9519,C -1.6014,E1 24.9786,E2 712.5547} C_DIS
LIN {X -14.7856,Y 133.6796,Z 153,A 92.0844,B 24.9519,C -1.6022,E1 24.9838,E2 714.4442} C_DIS
LIN {X -11.0162,Y 134.0427,Z 153,A 90.4633,B 24.9519,C -1.6026,E1 24.9883,E2 716.0652} C_DIS
LIN {X -6.7633,Y 134.3241,Z 153,A 88.6621,B 24.9518,C -1.604,E1 24.9933,E2 717.8635} C_DIS
LIN {X -2.4039,Y 134.473,Z 153,A 86.8298,B 24.9517,C -1.6059,E1 24.9984,E2 719.6916} C_DIS
LIN {X 1.621,Y 134.486,Z 153,A 85.0464,B 24.9519,C -1.6026,E1 25.0034,E2 721.4826} C_DIS
LIN {X 5.5392,Y 134.3805,Z 153,A 83.3523,B 24.9519,C -1.6015,E1 25.0082,E2 723.1789} C_DIS
LIN {X 9.746,Y 134.1407,Z 153,A 81.6562,B 24.9516,C -1.6066,E1 25.0129,E2 724.8622} C_DIS
LIN {X 13.6478,Y 133.802,Z 153,A 79.9083,B 24.9519,C -1.6023,E1 25.0178,E2 726.6194} C_DIS
LIN {X 17.6787,Y 133.3274,Z 153,A 78.2586,B 24.9517,C -1.6061,E1 25.0223,E2 728.2588} C_DIS
LIN {X 21.908,Y 132.698,Z 153,A 76.4409,B 24.9517,C -1.6057,E1 25.0273,E2 730.0757} C_DIS
LIN {X 25.6646,Y 132.0233,Z 153,A 74.8618,B 24.9516,C -1.6075,E1 25.0316,E2 731.6488} C_DIS
LIN {X 29.4611,Y 131.2286,Z 153,A 73.1367,B 24.9519,C -1.6028,E1 25.0364,E2 733.3826} C_DIS
LIN {X 32.9761,Y 130.3888,Z 153,A 71.6446,B 24.9518,C -1.6044,E1 25.0404,E2 734.8688} C_DIS
LIN {X 36.4733,Y 129.4542,Z 153,A 70.1086,B 24.9518,C -1.6037,E1 25.0445,E2 736.404} C_DIS
LIN {X 40.2425,Y 128.3342,Z 153,A 68.4757,B 24.9518,C -1.6046,E1 25.0489,E2 738.0319} C_DIS
LIN {X 45.0862,Y 126.7129,Z 153,A 66.3701,B 24.9516,C -1.6064,E1 25.0544,E2 740.129} C_DIS
LIN {X 49.1446,Y 125.1943,Z 153,A 64.4527,B 24.952,C -1.6008,E1 25.0595,E2 742.0556} C_DIS
LIN {X 52.226,Y 123.9404,Z 153,A 63.0396,B 24.952,C -1.5995,E1 25.0631,E2 743.4685} C_DIS
LIN {X 55.2733,Y 122.6116,Z 153,A 61.6169,B 24.9522,C -1.5975,E1 25.0667,E2 744.8924} C_DIS
LIN {X 58.2012,Y 121.2488,Z 153,A 60.2029,B 24.9524,C -1.5938,E1 25.0703,E2 746.3116} C_DIS
LIN {X 61.3683,Y 119.6773,Z 153,A 58.7178,B 24.9524,C -1.5929,E1 25.074,E2 747.7947} C_DIS
LIN {X 64.7311,Y 117.8945,Z 153,A 56.9981,B 24.9529,C -1.5854,E1 25.0783,E2 749.5273} C_DIS
LIN {X 68.5976,Y 115.6874,Z 153,A 55.0857,B 24.9531,C -1.5817,E1 25.0829,E2 751.4425} C_DIS
LIN {X 72.21,Y 113.4678,Z 153,A 53.3351,B 24.9531,C -1.5818,E1 25.087,E2 753.1873} C_DIS
LIN {X 75.5825,Y 111.2494,Z 153,A 51.5829,B 24.9534,C -1.5772,E1 25.0911,E2 754.9446} C_DIS
LIN {X 79.0808,Y 108.7905,Z 153,A 49.8061,B 24.9534,C -1.5764,E1 25.0951,E2 756.7171} C_DIS
LIN {X 82.6824,Y 106.0795,Z 153,A 47.8668,B 24.9537,C -1.5718,E1 25.0994,E2 758.6601} C_DIS
LIN {X 86.1175,Y 103.3105,Z 153,A 45.9832,B 24.9539,C -1.568,E1 25.1035,E2 760.5456} C_DIS
LIN {X 89.4815,Y 100.4105,Z 153,A 44.1043,B 24.9541,C -1.5648,E1 25.1075,E2 762.4245} C_DIS
LIN {X 92.7045,Y 97.4426,Z 153,A 42.2285,B 24.9544,C -1.5604,E1 25.1113,E2 764.3031} C_DIS
LIN {X 95.9268,Y 94.2717,Z 153,A 40.3778,B 24.9544,C -1.5602,E1 25.1149,E2 766.1463} C_DIS
LIN {X 98.8993,Y 91.1485,Z 153,A 38.4905,B 24.9548,C -1.5533,E1 25.1186,E2 768.0417} C_DIS
LIN {X 101.9549,Y 87.7171,Z 153,A 36.5725,B 24.9549,C -1.5509,E1 25.1221,E2 769.9569} C_DIS
LIN {X 104.7959,Y 84.3026,Z 153,A 34.73,B 24.955,C -1.549,E1 25.1253,E2 771.7953} C_DIS
LIN {X 107.4677,Y 80.8692,Z 153,A 32.8825,B 24.9553,C -1.5447,E1 25.1285,E2 773.6442} C_DIS
LIN {X 110.0688,Y 77.2919,Z 153,A 31.0303,B 24.9555,C -1.5416,E1 25.1315,E2 775.4947} C_DIS
LIN {X 112.4666,Y 73.7592,Z 153,A 29.1861,B 24.9558,C -1.5354,E1 25.1344,E2 777.3444} C_DIS
LIN {X 114.8552,Y 69.9824,Z 153,A 27.2561,B 24.9562,C -1.5288,E1 25.1372,E2 779.2802} C_DIS
LIN {X 117.0492,Y 66.2477,Z 153,A 25.3969,B 24.9565,C -1.5229,E1 25.1398,E2 781.1436} C_DIS
LIN {X 119.107,Y 62.4668,Z 153,A 23.7073,B 24.9564,C -1.5257,E1 25.142,E2 782.8176} C_DIS
LIN {X 120.5935,Y 59.5466,Z 153,A 22.2729,B 24.9567,C -1.5196,E1 25.1438,E2 784.2589} C_DIS
LIN {X 122.2742,Y 56.0163,Z 153,A 20.6687,B 24.9568,C -1.5181,E1 25.1457,E2 785.8579} C_DIS
LIN {X 123.4577,Y 53.3554,Z 153,A 19.3823,B 24.9572,C -1.512,E1 25.1472,E2 787.1519} C_DIS
LIN {X 124.9323,Y 49.8074,Z 153,A 17.8195,B 24.9572,C -1.5111,E1 25.1488,E2 788.7079} C_DIS
LIN {X 126.029,Y 46.9612,Z 153,A 16.4975,B 24.9575,C -1.506,E1 25.1501,E2 790.0347} C_DIS
LIN {X 127.3142,Y 43.3618,Z 153,A 14.8277,B 24.9579,C -1.4987,E1 25.1517,E2 791.7124} C_DIS
LIN {X 129.334,Y 36.9033,Z 153,A 12.08,B 24.958,C -1.4972,E1 25.1539,E2 794.4479} C_DIS
LIN {X 130.0592,Y 34.2549,Z 153,A 10.9059,B 24.9582,C -1.4933,E1 25.1547,E2 795.6244} C_DIS
LIN {X 130.8076,Y 31.2743,Z 153,A 9.6128,B 24.9584,C -1.4901,E1 25.1556,E2 796.9177} C_DIS
LIN {X 131.4994,Y 28.224,Z 153,A 8.2349,B 24.9588,C -1.4833,E1 25.1564,E2 798.3035} C_DIS
LIN {X 132.1633,Y 24.9327,Z 153,A 6.7762,B 24.9591,C -1.4771,E1 25.1572,E2 799.7683} C_DIS
LIN {X 132.8803,Y 20.7734,Z 153,A 5.0121,B 24.9593,C -1.4732,E1 25.158,E2 801.5313} C_DIS
LIN {X 133.4209,Y 16.9653,Z 153,A 3.4194,B 24.9595,C -1.4704,E1 25.1586,E2 803.1212} C_DIS
LIN {X 133.8705,Y 12.9378,Z 153,A 1.6634,B 24.9599,C -1.4631,E1 25.1591,E2 804.8839} C_DIS
LIN {X 134.1539,Y 9.5651,Z 153,A 0.2848,B 24.9599,C -1.4619,E1 25.1594,E2 806.2572} C_DIS
LIN {X 134.3772,Y 5.6244,Z 153,A -1.4818,B 24.9605,C -1.4516,E1 25.1597,E2 808.0376} C_DIS
LIN {X 134.4806,Y 1.9455,Z 153,A -2.9892,B 24.9606,C -1.4498,E1 25.1597,E2 809.5403} C_DIS
LIN {X 134.4766,Y -2.1846,Z 153,A -4.7842,B 24.961,C -1.442,E1 25.1597,E2 811.343} C_DIS
LIN {X 134.3301,Y -6.6451,Z 153,A -6.6224,B 24.9612,C -1.4392,E1 25.1595,E2 813.1768} C_DIS
LIN {X 134.125,Y -9.9613,Z 153,A -8.0169,B 24.9614,C -1.4356,E1 25.1593,E2 814.5714} C_DIS
LIN {X 133.7659,Y -13.9838,Z 153,A -9.7536,B 24.9617,C -1.429,E1 25.1588,E2 816.3134} C_DIS
LIN {X 133.3625,Y -17.4103,Z 153,A -11.1828,B 24.9619,C -1.4264,E1 25.1583,E2 817.7403} C_DIS
LIN {X 132.8359,Y -21.0602,Z 153,A -12.8102,B 24.9623,C -1.418,E1 25.1576,E2 819.3778} C_DIS
LIN {X 132.125,Y -25.1328,Z 153,A -14.5413,B 24.9626,C -1.4139,E1 25.1568,E2 821.1085} C_DIS
LIN {X 131.2817,Y -29.2284,Z 153,A -16.4136,B 24.9631,C -1.403,E1 25.1557,E2 822.9957} C_DIS
LIN {X 130.3589,Y -33.0938,Z 153,A -17.9445,B 24.9629,C -1.4065,E1 25.1547,E2 824.5094} C_DIS
LIN {X 129.3994,Y -36.6694,Z 153,A -19.452,B 24.963,C -1.4053,E1 25.1535,E2 826.0111} C_DIS
LIN {X 128.4813,Y -39.7662,Z 153,A -20.841,B 24.9633,C -1.4001,E1 25.1524,E2 827.4045} C_DIS
LIN {X 127.4799,Y -42.8678,Z 153,A -22.2089,B 24.9635,C -1.3968,E1 25.1512,E2 828.7725} C_DIS
LIN {X 126.4603,Y -45.7867,Z 153,A -23.5467,B 24.9637,C -1.3914,E1 25.15,E2 830.1153} C_DIS
LIN {X 125.1988,Y -49.133,Z 153,A -25.0423,B 24.9639,C -1.3881,E1 25.1485,E2 831.6104} C_DIS
LIN {X 123.9653,Y -52.1664,Z 153,A -26.4214,B 24.9641,C -1.3846,E1 25.147,E2 832.9902} C_DIS
LIN {X 122.7026,Y -55.0698,Z 153,A -27.7867,B 24.9644,C -1.3795,E1 25.1455,E2 834.3601} C_DIS
LIN {X 121.2747,Y -58.1469,Z 153,A -29.2688,B 24.9647,C -1.373,E1 25.1437,E2 835.8496} C_DIS
LIN {X 119.6119,Y -61.4967,Z 153,A -30.938,B 24.9652,C -1.3638,E1 25.1416,E2 837.5314} C_DIS
LIN {X 117.5452,Y -65.3626,Z 153,A -32.7723,B 24.9654,C -1.36,E1 25.1391,E2 839.3651} C_DIS
LIN {X 115.4076,Y -69.067,Z 153,A -34.6003,B 24.9656,C -1.3543,E1 25.1365,E2 841.1973} C_DIS
LIN {X 112.9757,Y -72.9773,Z 153,A -36.5448,B 24.9659,C -1.3495,E1 25.1336,E2 843.1432} C_DIS
LIN {X 110.4633,Y -76.7266,Z 153,A -38.4223,B 24.966,C -1.3465,E1 25.1307,E2 845.0185} C_DIS
LIN {X 108.0647,Y -80.07,Z 153,A -40.1206,B 24.9661,C -1.3446,E1 25.1279,E2 846.7131} C_DIS
LIN {X 105.685,Y -83.1854,Z 153,A -41.77,B 24.9663,C -1.3412,E1 25.1251,E2 848.3629} C_DIS
LIN {X 103.157,Y -86.3004,Z 153,A -43.557,B 24.9668,C -1.3322,E1 25.1219,E2 850.1627} C_DIS
LIN {X 100.1975,Y -89.7193,Z 153,A -45.4074,B 24.9668,C -1.3313,E1 25.1185,E2 852.0069} C_DIS
LIN {X 97.4401,Y -92.7071,Z 153,A -47.2022,B 24.9672,C -1.3234,E1 25.115,E2 853.8125} C_DIS
LIN {X 94.2754,Y -95.9232,Z 153,A -49.1002,B 24.9674,C -1.3199,E1 25.1113,E2 855.7107} C_DIS
LIN {X 90.9001,Y -99.1277,Z 153,A -51.0458,B 24.9675,C -1.3171,E1 25.1073,E2 857.6549} C_DIS
LIN {X 87.5233,Y -102.1218,Z 153,A -52.9778,B 24.9678,C -1.3121,E1 25.1032,E2 859.5912} C_DIS
LIN {X 84.1046,Y -104.9556,Z 153,A -54.8267,B 24.9678,C -1.3101,E1 25.0992,E2 861.4377} C_DIS
LIN {X 80.68,Y -107.6104,Z 153,A -56.723,B 24.9682,C -1.3033,E1 25.095,E2 863.3432} C_DIS
LIN {X 77.2424,Y -110.1037,Z 153,A -58.3201,B 24.9678,C -1.3111,E1 25.0914,E2 864.9162} C_DIS
LIN {X 74.7452,Y -111.8135,Z 153,A -59.7417,B 24.9683,C -1.3012,E1 25.0881,E2 866.3564} C_DIS
LIN {X 71.3735,Y -113.9959,Z 153,A -61.4822,B 24.9685,C -1.2962,E1 25.084,E2 868.1031} C_DIS
LIN {X 67.6373,Y -116.2514,Z 153,A -63.3589,B 24.9687,C -1.2918,E1 25.0795,E2 869.9845} C_DIS
LIN {X 64.0541,Y -118.2639,Z 153,A -65.1162,B 24.9689,C -1.2883,E1 25.0752,E2 871.745} C_DIS
LIN {X 60.8446,Y -119.9439,Z 153,A -66.5413,B 24.9687,C -1.2921,E1 25.0717,E2 873.1572} C_DIS
LIN {X 57.925,Y -121.3807,Z 153,A -67.9321,B 24.9689,C -1.2895,E1 25.0682,E2 874.5503} C_DIS
LIN {X 54.815,Y -122.8166,Z 153,A -69.3728,B 24.9689,C -1.2882,E1 25.0645,E2 875.9905} C_DIS
LIN {X 51.5549,Y -124.2206,Z 153,A -70.857,B 24.9689,C -1.2875,E1 25.0607,E2 877.473} C_DIS
LIN {X 48.2624,Y -125.5372,Z 153,A -72.3438,B 24.9689,C -1.2866,E1 25.0568,E2 878.9586} C_DIS
LIN {X 45.135,Y -126.6953,Z 153,A -73.7542,B 24.9691,C -1.2852,E1 25.0531,E2 880.3692} C_DIS
LIN {X 42.223,Y -127.6946,Z 153,A -75.1371,B 24.9693,C -1.2797,E1 25.0494,E2 881.7625} C_DIS
LIN {X 36.9756,Y -129.3137,Z 153,A -77.407,B 24.9693,C -1.2807,E1 25.0434,E2 884.0262} C_DIS
LIN {X 33.0084,Y -130.3806,Z 153,A -79.2153,B 24.9695,C -1.2757,E1 25.0385,E2 885.8434} C_DIS
LIN {X 28.7795,Y -131.3794,Z 153,A -81.1033,B 24.9697,C -1.2719,E1 25.0333,E2 887.7377} C_DIS
LIN {X 25.0283,Y -132.145,Z 153,A -82.6169,B 24.9695,C -1.2768,E1 25.0292,E2 889.238} C_DIS
LIN {X 22.1229,Y -132.6621,Z 153,A -83.9261,B 24.9696,C -1.273,E1 25.0256,E2 890.5548} C_DIS
LIN {X 18.4226,Y -133.2278,Z 153,A -85.5619,B 24.9698,C -1.2697,E1 25.021,E2 892.197} C_DIS
LIN {X 14.4479,Y -133.7159,Z 153,A -87.2134,B 24.9698,C -1.2715,E1 25.0165,E2 893.8429} C_DIS
LIN {X 11.2538,Y -134.0226,Z 153,A -88.589,B 24.9698,C -1.2704,E1 25.0126,E2 895.2205} C_DIS
LIN {X 7.3062,Y -134.2968,Z 153,A -90.3595,B 24.97,C -1.2651,E1 25.0077,E2 897.0027} C_DIS
LIN {X 3.2609,Y -134.4556,Z 153,A -91.9876,B 24.9698,C -1.2696,E1 25.0032,E2 898.6197} C_DIS
LIN {X 0.9478,Y -134.4897,Z 153,A -92.8917,B 24.9696,C -1.2737,E1 25.0007,E2 899.514} C_DIS
Enddeposition()
LIN {X 0.9478,Y -134.4897,Z 153,A -92.8917,B 24.9696,C -1.2737,E1 25.0007,E2 899.514} C_DIS
Startdeposition()
$VEL.CP = VEL_PRINT
LIN {X 1.5029,Y -133.5476,Z 153,A -91.8731,B 24.645,C -1.2631,E1 24.6789,E2 898.4788} C_DIS
LIN {X 5.3468,Y -133.4471,Z 153,A -90.3237,B 24.6452,C -1.2584,E1 24.6832,E2 896.941} C_DIS
LIN {X 9.7495,Y -133.1977,Z 153,A -88.457,B 24.6452,C -1.2579,E1 24.6884,E2 895.0762} C_DIS
LIN {X 13.6763,Y -132.8533,Z 153,A -86.6785,B 24.645,C -1.2634,E1 24.6934,E2 893.2856} C_DIS
LIN {X 17.4341,Y -132.4112,Z 153,A -85.1477,B 24.6452,C -1.2596,E1 24.6976,E2 891.7653} C_DIS
LIN {X 21.203,Y -131.8624,Z 153,A -83.3814,B 24.6448,C -1.2678,E1 24.7025,E2 889.981} C_DIS
LIN {X 25.3595,Y -131.1244,Z 153,A -81.7477,B 24.6452,C -1.2599,E1 24.7069,E2 888.3681} C_DIS
LIN {X 28.5856,Y -130.4594,Z 153,A -80.299,B 24.645,C -1.2631,E1 24.7109,E2 886.9137} C_DIS
LIN {X 32.6246,Y -129.508,Z 153,A -78.412,B 24.6447,C -1.2705,E1 24.7161,E2 885.0115} C_DIS
LIN {X 36.7501,Y -128.4005,Z 153,A -76.7133,B 24.6449,C -1.2654,E1 24.7206,E2 883.328} C_DIS
LIN {X 39.5728,Y -127.5573,Z 153,A -75.3544,B 24.6446,C -1.272,E1 24.7243,E2 881.9558} C_DIS
LIN {X 43.8015,Y -126.1666,Z 153,A -73.5468,B 24.6447,C -1.269,E1 24.729,E2 880.159} C_DIS
LIN {X 46.9844,Y -125.0163,Z 153,A -72.0857,B 24.6447,C -1.2714,E1 24.7328,E2 878.6951} C_DIS
LIN {X 50.1228,Y -123.7915,Z 153,A -70.6341,B 24.6445,C -1.2738,E1 24.7366,E2 877.2411} C_DIS
LIN {X 53.2458,Y -122.4807,Z 153,A -69.2124,B 24.6445,C -1.2743,E1 24.7403,E2 875.8216} C_DIS
LIN {X 56.2388,Y -121.1355,Z 153,A -67.7925,B 24.6443,C -1.2772,E1 24.7439,E2 874.3984} C_DIS
LIN {X 59.2814,Y -119.6759,Z 153,A -66.3732,B 24.6443,C -1.2781,E1 24.7474,E2 872.9808} C_DIS
LIN {X 62.1508,Y -118.211,Z 153,A -65.0076,B 24.6443,C -1.2796,E1 24.7508,E2 871.6155} C_DIS
LIN {X 65.5823,Y -116.3446,Z 153,A -62.8932,B 24.6429,C -1.3064,E1 24.7561,E2 869.4433} C_DIS
LIN {X 68.9208,Y -114.3986,Z 153,A -61.6454,B 24.6438,C -1.2872,E1 24.759,E2 868.2453} C_DIS
LIN {X 74.7617,Y -110.6697,Z 153,A -58.8059,B 24.6439,C -1.2858,E1 24.7656,E2 865.4186} C_DIS
LIN {X 78.8757,Y -107.7764,Z 153,A -56.6045,B 24.6436,C -1.2927,E1 24.7707,E2 863.2085} C_DIS
LIN {X 81.5888,Y -105.7376,Z 153,A -55.0024,B 24.643,C -1.3038,E1 24.7742,E2 861.5857} C_DIS
LIN {X 84.9197,Y -103.0817,Z 153,A -53.1515,B 24.6428,C -1.3092,E1 24.7783,E2 859.729} C_DIS
LIN {X 88.3656,Y -100.1429,Z 153,A -51.2718,B 24.6428,C -1.3103,E1 24.7822,E2 857.8542} C_DIS
LIN {X 91.4817,Y -97.3048,Z 153,A -49.4327,B 24.6424,C -1.3164,E1 24.786,E2 856.0083} C_DIS
LIN {X 94.7584,Y -94.1166,Z 153,A -47.5061,B 24.6423,C -1.3193,E1 24.7898,E2 854.0828} C_DIS
LIN {X 97.8989,Y -90.8457,Z 153,A -45.5911,B 24.6421,C -1.3226,E1 24.7935,E2 852.1684} C_DIS
LIN {X 100.8669,Y -87.5389,Z 153,A -43.6435,B 24.6417,C -1.3299,E1 24.7971,E2 850.2123} C_DIS
LIN {X 103.7043,Y -84.1585,Z 153,A -41.7445,B 24.6414,C -1.3353,E1 24.8005,E2 848.3093} C_DIS
LIN {X 107.5407,Y -79.1966,Z 153,A -38.9316,B 24.6407,C -1.3495,E1 24.8053,E2 845.4761} C_DIS
LIN {X 110.6998,Y -74.7173,Z 153,A -36.6374,B 24.6405,C -1.353,E1 24.8089,E2 843.185} C_DIS
LIN {X 112.9019,Y -71.346,Z 153,A -35.0492,B 24.6407,C -1.3503,E1 24.8113,E2 841.6113} C_DIS
LIN {X 115.1904,Y -67.5888,Z 153,A -33.1833,B 24.6405,C -1.3547,E1 24.8139,E2 839.7447} C_DIS
LIN {X 117.4249,Y -63.6288,Z 153,A -31.2366,B 24.6402,C -1.3603,E1 24.8166,E2 837.7949} C_DIS
LIN {X 119.1212,Y -60.3884,Z 153,A -29.7783,B 24.6402,C -1.359,E1 24.8184,E2 836.3477} C_DIS
LIN {X 120.6667,Y -57.2384,Z 153,A -28.3032,B 24.6401,C -1.3619,E1 24.8202,E2 834.8736} C_DIS
LIN {X 121.9554,Y -54.4377,Z 153,A -26.9578,B 24.6398,C -1.3673,E1 24.8218,E2 833.5228} C_DIS
LIN {X 123.3305,Y -51.2466,Z 153,A -25.4449,B 24.6395,C -1.3732,E1 24.8234,E2 832.0042} C_DIS
LIN {X 124.8988,Y -47.2981,Z 153,A -23.56,B 24.639,C -1.3824,E1 24.8253,E2 830.1081} C_DIS
LIN {X 126.2186,Y -43.6517,Z 153,A -22.0362,B 24.6391,C -1.3799,E1 24.8267,E2 828.5988} C_DIS
LIN {X 127.2813,Y -40.4489,Z 153,A -20.6078,B 24.639,C -1.3835,E1 24.828,E2 827.1701} C_DIS
LIN {X 128.2219,Y -37.3601,Z 153,A -19.2128,B 24.6387,C -1.3885,E1 24.8291,E2 825.7712} C_DIS
LIN {X 129.2404,Y -33.6767,Z 153,A -17.4564,B 24.6381,C -1.4003,E1 24.8304,E2 823.9969} C_DIS
LIN {X 130.193,Y -29.7726,Z 153,A -15.8736,B 24.6381,C -1.3981,E1 24.8314,E2 822.4286} C_DIS
LIN {X 130.9578,Y -26.2082,Z 153,A -14.1899,B 24.6375,C -1.4099,E1 24.8323,E2 820.7268} C_DIS
LIN {X 131.7312,Y -21.9895,Z 153,A -12.4871,B 24.6376,C -1.4083,E1 24.8331,E2 819.0379} C_DIS
LIN {X 132.2421,Y -18.6743,Z 153,A -11.0366,B 24.6373,C -1.4137,E1 24.8337,E2 817.5833} C_DIS
LIN {X 132.7692,Y -14.4583,Z 153,A -9.2394,B 24.6371,C -1.4183,E1 24.8343,E2 815.7859} C_DIS
LIN {X 133.1008,Y -10.996,Z 153,A -7.6987,B 24.6367,C -1.4259,E1 24.8347,E2 814.2362} C_DIS
LIN {X 133.3791,Y -6.8361,Z 153,A -5.9867,B 24.6366,C -1.4276,E1 24.835,E2 812.5306} C_DIS
LIN {X 133.5155,Y -3.245,Z 153,A -4.3884,B 24.6361,C -1.4358,E1 24.8351,E2 810.9223} C_DIS
LIN {X 133.5502,Y 1.0423,Z 153,A -2.5595,B 24.6358,C -1.4413,E1 24.8351,E2 809.0914} C_DIS
LIN {X 133.4487,Y 5.3062,Z 153,A -0.8121,B 24.6358,C -1.4428,E1 24.835,E2 807.351} C_DIS
LIN {X 133.2421,Y 9.1415,Z 153,A 0.9087,B 24.6352,C -1.4522,E1 24.8347,E2 805.6181} C_DIS
LIN {X 132.9224,Y 12.9758,Z 153,A 2.467,B 24.6352,C -1.4525,E1 24.8343,E2 804.0685} C_DIS
LIN {X 132.5574,Y 16.2922,Z 153,A 3.8203,B 24.6352,C -1.4528,E1 24.8338,E2 802.7224} C_DIS
LIN {X 132.1407,Y 19.3839,Z 153,A 5.3438,B 24.6344,C -1.4674,E1 24.8332,E2 801.1732} C_DIS
LIN {X 131.4759,Y 23.4681,Z 153,A 6.9625,B 24.6346,C -1.4645,E1 24.8325,E2 799.5712} C_DIS
LIN {X 130.8273,Y 26.8495,Z 153,A 8.4433,B 24.6343,C -1.4694,E1 24.8317,E2 798.0874} C_DIS
LIN {X 130.09,Y 30.2236,Z 153,A 9.861,B 24.6343,C -1.4706,E1 24.8308,E2 796.6754} C_DIS
LIN {X 129.3934,Y 33.0761,Z 153,A 11.2101,B 24.6337,C -1.4795,E1 24.8299,E2 795.3129} C_DIS
LIN {X 127.9385,Y 38.3271,Z 153,A 13.4636,B 24.6336,C -1.4821,E1 24.8282,E2 793.0663} C_DIS
LIN {X 126.988,Y 41.3671,Z 153,A 14.8244,B 24.6334,C -1.486,E1 24.827,E2 791.704} C_DIS
LIN {X 126.0674,Y 44.0878,Z 153,A 16.1564,B 24.6328,C -1.4953,E1 24.8258,E2 790.3575} C_DIS
LIN {X 124.4926,Y 48.3548,Z 153,A 18.0197,B 24.6328,C -1.4963,E1 24.8239,E2 788.5022} C_DIS
LIN {X 123.1901,Y 51.5829,Z 153,A 19.4946,B 24.6326,C -1.4997,E1 24.8224,E2 787.0273} C_DIS
LIN {X 121.8016,Y 54.7814,Z 153,A 21.0017,B 24.6323,C -1.5047,E1 24.8207,E2 785.5167} C_DIS
LIN {X 120.3667,Y 57.8664,Z 153,A 22.433,B 24.6321,C -1.5074,E1 24.8189,E2 784.0869} C_DIS
LIN {X 118.6803,Y 61.2543,Z 153,A 24.2084,B 24.6314,C -1.5203,E1 24.8167,E2 782.2901} C_DIS
LIN {X 116.304,Y 65.6546,Z 153,A 26.2666,B 24.6314,C -1.5215,E1 24.8139,E2 780.24} C_DIS
LIN {X 114.0563,Y 69.4867,Z 153,A 28.1665,B 24.631,C -1.5264,E1 24.8112,E2 778.3384} C_DIS
LIN {X 111.7559,Y 73.129,Z 153,A 30.0278,B 24.6307,C -1.532,E1 24.8084,E2 776.4731} C_DIS
LIN {X 109.3038,Y 76.7453,Z 153,A 31.8416,B 24.6307,C -1.5336,E1 24.8055,E2 774.6646} C_DIS
LIN {X 106.8017,Y 80.1909,Z 153,A 33.7059,B 24.6302,C -1.5403,E1 24.8024,E2 772.7934} C_DIS
LIN {X 103.9997,Y 83.7923,Z 153,A 35.6144,B 24.6302,C -1.5424,E1 24.7991,E2 770.8889} C_DIS
LIN {X 101.289,Y 87.0496,Z 153,A 37.4254,B 24.6299,C -1.5464,E1 24.7958,E2 769.0768} C_DIS
LIN {X 98.5151,Y 90.1772,Z 153,A 39.2378,B 24.6296,C -1.5516,E1 24.7924,E2 767.2603} C_DIS
LIN {X 95.489,Y 93.3754,Z 153,A 41.1014,B 24.6294,C -1.5544,E1 24.7888,E2 765.398} C_DIS
LIN {X 92.4025,Y 96.4307,Z 153,A 42.9664,B 24.6291,C -1.5585,E1 24.7851,E2 763.5311} C_DIS
LIN {X 89.2125,Y 99.3893,Z 153,A 44.8209,B 24.629,C -1.5618,E1 24.7812,E2 761.6764} C_DIS
LIN {X 85.7186,Y 102.4179,Z 153,A 46.7888,B 24.6288,C -1.5649,E1 24.7771,E2 759.7089} C_DIS
LIN {X 82.2209,Y 105.2469,Z 153,A 48.72,B 24.6286,C -1.5686,E1 24.7728,E2 757.7761} C_DIS
LIN {X 78.6815,Y 107.9187,Z 153,A 50.6498,B 24.6283,C -1.5735,E1 24.7685,E2 755.8416} C_DIS
LIN {X 75.0722,Y 110.4595,Z 153,A 52.522,B 24.6281,C -1.5756,E1 24.7642,E2 753.9709} C_DIS
LIN {X 71.346,Y 112.9019,Z 153,A 54.4066,B 24.6281,C -1.5772,E1 24.7598,E2 752.0885} C_DIS
LIN {X 67.7018,Y 115.1241,Z 153,A 56.2089,B 24.628,C -1.5785,E1 24.7555,E2 750.2889} C_DIS
LIN {X 63.8001,Y 117.3314,Z 153,A 58.1503,B 24.6277,C -1.5822,E1 24.7507,E2 748.3444} C_DIS
LIN {X 60.3935,Y 119.1185,Z 153,A 59.7101,B 24.6279,C -1.5796,E1 24.7469,E2 746.7951} C_DIS
LIN {X 57.1741,Y 120.6975,Z 153,A 61.1907,B 24.6279,C -1.5785,E1 24.7432,E2 745.3212} C_DIS
LIN {X 54.342,Y 121.9982,Z 153,A 62.5604,B 24.6278,C -1.5818,E1 24.7397,E2 743.947} C_DIS
LIN {X 51.3987,Y 123.267,Z 153,A 63.9471,B 24.6276,C -1.584,E1 24.7361,E2 742.5585} C_DIS
LIN {X 48.1967,Y 124.554,Z 153,A 65.4301,B 24.6276,C -1.5856,E1 24.7322,E2 741.0749} C_DIS
LIN {X 44.5539,Y 125.9054,Z 153,A 67.4,B 24.6265,C -1.6031,E1 24.727,E2 739.0673} C_DIS
LIN {X 41.3499,Y 126.9935,Z 153,A 68.485,B 24.6276,C -1.585,E1 24.7242,E2 738.0276} C_DIS
LIN {X 38.4949,Y 127.8872,Z 153,A 69.783,B 24.6275,C -1.5868,E1 24.7207,E2 736.7277} C_DIS
LIN {X 35.6882,Y 128.6975,Z 153,A 71.0458,B 24.6274,C -1.5882,E1 24.7173,E2 735.4636} C_DIS
LIN {X 32.4147,Y 129.5612,Z 153,A 72.6311,B 24.6269,C -1.5961,E1 24.713,E2 733.862} C_DIS
LIN {X 28.3765,Y 130.5046,Z 153,A 74.3186,B 24.6271,C -1.5922,E1 24.7084,E2 732.1859} C_DIS
LIN {X 24.9994,Y 131.1933,Z 153,A 75.758,B 24.6272,C -1.5909,E1 24.7045,E2 730.7515} C_DIS
LIN {X 21.2336,Y 131.8573,Z 153,A 77.5368,B 24.6267,C -1.5986,E1 24.6996,E2 728.9561} C_DIS
LIN {X 17.0792,Y 132.4577,Z 153,A 79.257,B 24.627,C -1.5949,E1 24.6948,E2 727.2462} C_DIS
LIN {X 12.865,Y 132.933,Z 153,A 81.045,B 24.627,C -1.5936,E1 24.6899,E2 725.4627} C_DIS
LIN {X 9.3352,Y 133.228,Z 153,A 82.6601,B 24.6267,C -1.5986,E1 24.6854,E2 723.8364} C_DIS
LIN {X 5.1308,Y 133.4556,Z 153,A 84.3513,B 24.6271,C -1.5926,E1 24.6807,E2 722.1601} C_DIS
LIN {X 1.5429,Y 133.547,Z 153,A 86.0389,B 24.6267,C -1.5999,E1 24.6759,E2 720.4551} C_DIS
LIN {X -2.662,Y 133.5283,Z 153,A 87.8033,B 24.6268,C -1.5975,E1 24.671,E2 718.6965} C_DIS
LIN {X -6.7735,Y 133.3822,Z 153,A 89.5018,B 24.6271,C -1.5935,E1 24.6663,E2 717.0072} C_DIS
LIN {X -11.0546,Y 133.0959,Z 153,A 91.3417,B 24.6271,C -1.5926,E1 24.6612,E2 715.1685} C_DIS
LIN {X -14.8896,Y 132.7228,Z 153,A 93.079,B 24.6269,C -1.596,E1 24.6563,E2 713.4221} C_DIS
LIN {X -18.9301,Y 132.2056,Z 153,A 94.717,B 24.6273,C -1.5894,E1 24.6518,E2 711.7987} C_DIS
LIN {X -22.5862,Y 131.6316,Z 153,A 96.2808,B 24.6274,C -1.587,E1 24.6475,E2 710.2392} C_DIS
LIN {X -26.4103,Y 130.9167,Z 153,A 98.061,B 24.6272,C -1.5913,E1 24.6426,E2 708.4467} C_DIS
LIN {X -30.25,Y 130.084,Z 153,A 99.6173,B 24.6277,C -1.5832,E1 24.6384,E2 706.9078} C_DIS
LIN {X -33.2143,Y 129.3583,Z 153,A 100.9537,B 24.6277,C -1.5832,E1 24.6348,E2 705.5693} C_DIS
LIN {X -37.0965,Y 128.2991,Z 153,A 102.7744,B 24.6275,C -1.5862,E1 24.6299,E2 703.7387} C_DIS
LIN {X -40.5379,Y 127.2529,Z 153,A 104.2393,B 24.6278,C -1.5805,E1 24.626,E2 702.285} C_DIS
LIN {X -43.7095,Y 126.1986,Z 153,A 105.668,B 24.628,C -1.5784,E1 24.6222,E2 700.8584} C_DIS
LIN {X -46.7459,Y 125.1056,Z 153,A 107.1439,B 24.6278,C -1.5812,E1 24.6183,E2 699.3728} C_DIS
LIN {X -50.3349,Y 123.7059,Z 153,A 108.7184,B 24.6282,C -1.5749,E1 24.6143,E2 697.8098} C_DIS
LIN {X -53.2817,Y 122.4652,Z 153,A 110.075,B 24.6283,C -1.5722,E1 24.6108,E2 696.4567} C_DIS
LIN {X -56.1684,Y 121.168,Z 153,A 111.469,B 24.6283,C -1.5719,E1 24.6073,E2 695.0599} C_DIS
LIN {X -59.4095,Y 119.6127,Z 153,A 113.0526,B 24.6283,C -1.5714,E1 24.6033,E2 693.4732} C_DIS
LIN {X -62.8841,Y 117.8253,Z 153,A 114.814,B 24.6283,C -1.5728,E1 24.5989,E2 691.7037} C_DIS
LIN {X -66.6685,Y 115.7258,Z 153,A 116.6571,B 24.6285,C -1.5688,E1 24.5944,E2 689.8647} C_DIS
LIN {X -70.305,Y 113.5534,Z 153,A 118.5021,B 24.6287,C -1.5667,E1 24.59,E2 688.0188} C_DIS
LIN {X -74.1424,Y 111.0855,Z 153,A 120.4501,B 24.6289,C -1.5624,E1 24.5855,E2 686.0747} C_DIS
LIN {X -77.8411,Y 108.5259,Z 153,A 122.7569,B 24.628,C -1.5771,E1 24.5802,E2 683.7245} C_DIS
LIN {X -81.1542,Y 106.0711,Z 153,A 124.163,B 24.6293,C -1.5554,E1 24.5771,E2 682.3656} C_DIS
LIN {X -84.0213,Y 103.815,Z 153,A 125.7044,B 24.6296,C -1.5507,E1 24.5738,E2 680.8295} C_DIS
LIN {X -87.0078,Y 101.325,Z 153,A 127.7353,B 24.6288,C -1.5648,E1 24.5694,E2 678.7567} C_DIS
LIN {X -89.9179,Y 98.7517,Z 153,A 129.5506,B 24.6286,C -1.5682,E1 24.5656,E2 676.9258} C_DIS
LIN {X -93.2852,Y 95.5775,Z 153,A 131.1005,B 24.6301,C -1.5419,E1 24.5626,E2 675.4326} C_DIS
LIN {X -96.2944,Y 92.5451,Z 153,A 133.5643,B 24.6286,C -1.5683,E1 24.5577,E2 672.8944} C_DIS
LIN {X -100.0267,Y 88.4971,Z 153,A 135.22,B 24.631,C -1.5276,E1 24.5548,E2 671.3295} C_DIS
LIN {X -102.6505,Y 85.4404,Z 153,A 137.0629,B 24.631,C -1.5286,E1 24.5514,E2 669.4755} C_DIS
LIN {X -105.4439,Y 81.9677,Z 153,A 138.9379,B 24.6313,C -1.5216,E1 24.5482,E2 667.6084} C_DIS
LIN {X -107.9926,Y 78.5795,Z 153,A 140.8123,B 24.6314,C -1.5193,E1 24.5451,E2 665.7304} C_DIS
LIN {X -110.6465,Y 74.796,Z 153,A 142.7834,B 24.6318,C -1.5131,E1 24.542,E2 663.7643} C_DIS
LIN {X -112.9038,Y 71.343,Z 153,A 144.5579,B 24.6321,C -1.5083,E1 24.5393,E2 661.9924} C_DIS
LIN {X -115.2665,Y 67.4594,Z 153,A 146.4992,B 24.6324,C -1.5021,E1 24.5365,E2 660.0558} C_DIS
LIN {X -117.3135,Y 63.833,Z 153,A 148.7613,B 24.6314,C -1.5199,E1 24.5334,E2 657.7386} C_DIS
LIN {X -119.3901,Y 59.8601,Z 153,A 150.7369,B 24.6316,C -1.5166,E1 24.5309,E2 655.7602} C_DIS
LIN {X -121.353,Y 55.7684,Z 153,A 152.0024,B 24.6338,C -1.4776,E1 24.5296,E2 654.5818} C_DIS
LIN {X -122.9828,Y 52.0792,Z 153,A 153.7971,B 24.634,C -1.4753,E1 24.5275,E2 652.7825} C_DIS
LIN {X -124.5238,Y 48.2744,Z 153,A 155.6467,B 24.634,C -1.4741,E1 24.5256,E2 650.9255} C_DIS
LIN {X -125.7504,Y 44.9837,Z 153,A 157.1561,B 24.6343,C -1.4695,E1 24.5242,E2 649.4185} C_DIS
LIN {X -127.4878,Y 39.7984,Z 153,A 159.6049,B 24.6344,C -1.4669,E1 24.5221,E2 646.9618} C_DIS
LIN {X -128.4739,Y 36.4877,Z 153,A 161.0145,B 24.6349,C -1.4586,E1 24.521,E2 645.5638} C_DIS
LIN {X -129.3434,Y 33.2729,Z 153,A 162.5116,B 24.6349,C -1.4573,E1 24.5199,E2 644.061} C_DIS
LIN {X -131.0236,Y 25.8848,Z 153,A 166.2947,B 24.6341,C -1.4724,E1 24.5177,E2 640.2188} C_DIS
LIN {X -131.8414,Y 21.329,Z 153,A 167.6555,B 24.6362,C -1.4357,E1 24.5171,E2 638.9385} C_DIS
LIN {X -132.4957,Y 16.7893,Z 153,A 169.8122,B 24.636,C -1.4383,E1 24.5162,E2 636.7623} C_DIS
LIN {X -132.9494,Y 12.6942,Z 153,A 171.5056,B 24.6365,C -1.4289,E1 24.5158,E2 635.0813} C_DIS
LIN {X -133.2817,Y 8.5318,Z 153,A 173.3264,B 24.6368,C -1.4244,E1 24.5154,E2 633.2602} C_DIS
LIN {X -133.4666,Y 4.8474,Z 153,A 175.0089,B 24.6368,C -1.424,E1 24.5152,E2 631.5684} C_DIS
LIN {X -133.5516,Y 0.7655,Z 153,A 176.6861,B 24.6373,C -1.4147,E1 24.5152,E2 629.9036} C_DIS
LIN {X -133.5064,Y -3.5721,Z 153,A 178.5733,B 24.6376,C -1.4098,E1 24.5152,E2 628.0165} C_DIS
LIN {X -133.3194,Y -7.9193,Z 153,A -179.558,B 24.6379,C -1.4038,E1 24.5155,E2 626.151} C_DIS
LIN {X -133.0309,Y -11.8245,Z 153,A -177.771,B 24.6379,C -1.4034,E1 24.5159,E2 624.3539} C_DIS
LIN {X -132.5175,Y -16.6233,Z 153,A -175.861,B 24.6387,C -1.389,E1 24.5165,E2 622.4672} C_DIS
LIN {X -131.9286,Y -20.7757,Z 153,A -173.8887,B 24.6385,C -1.3915,E1 24.5173,E2 620.4767} C_DIS
LIN {X -131.1734,Y -25.1035,Z 153,A -172.0855,B 24.6391,C -1.3816,E1 24.5182,E2 618.6868} C_DIS
LIN {X -130.3572,Y -29.0538,Z 153,A -170.3585,B 24.6394,C -1.3759,E1 24.5192,E2 616.9632} C_DIS
LIN {X -129.4633,Y -32.8004,Z 153,A -168.7008,B 24.6396,C -1.371,E1 24.5203,E2 615.3075} C_DIS
LIN {X -128.5675,Y -36.153,Z 153,A -167.2254,B 24.6399,C -1.3657,E1 24.5214,E2 613.8362} C_DIS
LIN {X -127.6177,Y -39.3755,Z 153,A -165.7367,B 24.6399,C -1.3635,E1 24.5226,E2 612.344} C_DIS
LIN {X -126.369,Y -43.218,Z 153,A -163.9033,B 24.64,C -1.363,E1 24.5243,E2 610.501} C_DIS
LIN {X -124.9569,Y -47.1431,Z 153,A -162.2183,B 24.6406,C -1.3526,E1 24.5259,E2 608.8316} C_DIS
LIN {X -123.7455,Y -50.2368,Z 153,A -160.7461,B 24.6406,C -1.3506,E1 24.5274,E2 607.3558} C_DIS
LIN {X -121.85,Y -54.6732,Z 153,A -158.6809,B 24.641,C -1.3443,E1 24.5297,E2 605.2943} C_DIS
LIN {X -120.3283,Y -57.9469,Z 153,A -157.1226,B 24.6412,C -1.3403,E1 24.5316,E2 603.737} C_DIS
LIN {X -118.5836,Y -61.4411,Z 153,A -155.3317,B 24.6412,C -1.3412,E1 24.5338,E2 601.9343} C_DIS
LIN {X -116.5193,Y -65.2716,Z 153,A -153.4541,B 24.6414,C -1.3365,E1 24.5364,E2 600.0579} C_DIS
LIN {X -114.1946,Y -69.2582,Z 153,A -151.4901,B 24.6417,C -1.3303,E1 24.5392,E2 598.0984} C_DIS
LIN {X -111.949,Y -72.8321,Z 153,A -149.6563,B 24.6419,C -1.3267,E1 24.5419,E2 596.2641} C_DIS
LIN {X -109.4472,Y -76.5409,Z 153,A -147.7114,B 24.6421,C -1.323,E1 24.545,E2 594.3183} C_DIS
LIN {X -106.8103,Y -80.1794,Z 153,A -145.2283,B 24.6409,C -1.3457,E1 24.5493,E2 591.7684} C_DIS
LIN {X -103.6458,Y -84.2304,Z 153,A -143.8559,B 24.6433,C -1.299,E1 24.5515,E2 590.502} C_DIS
LIN {X -101.8976,Y -86.3366,Z 153,A -142.3938,B 24.6427,C -1.3104,E1 24.5542,E2 589.0056} C_DIS
LIN {X -98.9934,Y -89.6515,Z 153,A -140.4875,B 24.6429,C -1.3068,E1 24.5577,E2 587.0993} C_DIS
LIN {X -95.796,Y -93.0605,Z 153,A -137.7283,B 24.6412,C -1.3401,E1 24.5633,E2 584.2478} C_DIS
LIN {X -91.4272,Y -97.3562,Z 153,A -136.0784,B 24.6439,C -1.2855,E1 24.5663,E2 582.7226} C_DIS
LIN {X -89.3532,Y -99.2632,Z 153,A -134.53,B 24.6432,C -1.2999,E1 24.5696,E2 581.133} C_DIS
LIN {X -86.6052,Y -101.6693,Z 153,A -133.0908,B 24.6437,C -1.2904,E1 24.5726,E2 579.711} C_DIS
LIN {X -83.378,Y -104.3324,Z 153,A -131.226,B 24.6437,C -1.2905,E1 24.5767,E2 577.8389} C_DIS
LIN {X -79.7748,Y -107.1124,Z 153,A -129.299,B 24.6439,C -1.2857,E1 24.581,E2 575.9164} C_DIS
LIN {X -76.1071,Y -109.749,Z 153,A -127.3787,B 24.6441,C -1.2815,E1 24.5853,E2 573.9995} C_DIS
LIN {X -72.6,Y -112.0997,Z 153,A -125.5296,B 24.6441,C -1.2804,E1 24.5896,E2 572.1467} C_DIS
LIN {X -68.822,Y -114.4584,Z 153,A -123.6127,B 24.6443,C -1.2778,E1 24.5942,E2 570.2301} C_DIS
LIN {X -65.0195,Y -116.6606,Z 153,A -121.6929,B 24.6443,C -1.2769,E1 24.5989,E2 568.3069} C_DIS
LIN {X -61.9088,Y -118.3381,Z 153,A -120.3072,B 24.6448,C -1.2683,E1 24.6023,E2 566.9379} C_DIS
LIN {X -58.9556,Y -119.8366,Z 153,A -118.8906,B 24.6448,C -1.2663,E1 24.6058,E2 565.5224} C_DIS
LIN {X -55.8644,Y -121.3086,Z 153,A -117.3835,B 24.6448,C -1.2664,E1 24.6096,E2 564.011} C_DIS
LIN {X -52.7756,Y -122.684,Z 153,A -115.9439,B 24.645,C -1.2643,E1 24.6133,E2 562.5732} C_DIS
LIN {X -49.587,Y -124.0074,Z 153,A -114.3938,B 24.6449,C -1.2663,E1 24.6173,E2 561.0148} C_DIS
LIN {X -44.3742,Y -125.9681,Z 153,A -112.1341,B 24.6453,C -1.2574,E1 24.6232,E2 558.7717} C_DIS
LIN {X -41.5579,Y -126.9251,Z 153,A -110.8069,B 24.6453,C -1.259,E1 24.6267,E2 557.4383} C_DIS
LIN {X -39.0567,Y -127.7152,Z 153,A -109.6703,B 24.6453,C -1.2587,E1 24.6298,E2 556.3003} C_DIS
LIN {X -35.8482,Y -128.6528,Z 153,A -108.1975,B 24.6452,C -1.2597,E1 24.6337,E2 554.8226} C_DIS
LIN {X -32.2579,Y -129.601,Z 153,A -106.6571,B 24.6454,C -1.256,E1 24.6379,E2 553.2888} C_DIS
LIN {X -28.8149,Y -130.4099,Z 153,A -105.0085,B 24.6451,C -1.262,E1 24.6424,E2 551.6236} C_DIS
LIN {X -25.1068,Y -131.1728,Z 153,A -103.4894,B 24.6454,C -1.256,E1 24.6466,E2 550.1174} C_DIS
LIN {X -21.7166,Y -131.7767,Z 153,A -101.9817,B 24.6454,C -1.257,E1 24.6507,E2 548.6057} C_DIS
LIN {X -17.5657,Y -132.394,Z 153,A -100.1805,B 24.6454,C -1.2567,E1 24.6557,E2 546.8038} C_DIS
LIN {X -14.101,Y -132.8076,Z 153,A -98.6882,B 24.6454,C -1.2562,E1 24.6598,E2 545.3116} C_DIS
LIN {X -9.9305,Y -133.1845,Z 153,A -96.8791,B 24.6454,C -1.2568,E1 24.6649,E2 543.5004} C_DIS
LIN {X -6.1184,Y -133.4152,Z 153,A -95.3077,B 24.6454,C -1.2534,E1 24.6692,E2 541.9367} C_DIS
LIN {X -2.396,Y -133.5328,Z 153,A -93.6445,B 24.6454,C -1.257,E1 24.6739,E2 540.2645} C_DIS
LIN {X 0.9452,Y -133.5492,Z 153,A -92.785,B 24.6467,C -1.2274,E1 24.6761,E2 539.476} C_DIS
Enddeposition()
LIN {X 0.9452,Y -133.5492,Z 153,A -92.785,B 24.6467,C -1.2274,E1 24.6761,E2 539.476} C_DIS
Startdeposition()
$VEL.CP = VEL_PRINT
LIN {X 0,Y -132.616,Z 153,A -92.9777,B 23.2979,C -0.9855,E1 23.3166,E2 540.0966} C_DIS
LIN {X -3.6596,Y -132.5635,Z 153,A -94.4469,B 23.2977,C -0.9907,E1 23.3125,E2 541.5528} C_DIS
LIN {X -7.4051,Y -132.4091,Z 153,A -96.0329,B 23.2977,C -0.9922,E1 23.3081,E2 543.1356} C_DIS
LIN {X -11.0016,Y -132.1568,Z 153,A -97.6344,B 23.2977,C -0.9901,E1 23.3036,E2 544.7429} C_DIS
LIN {X -14.4252,Y -131.8272,Z 153,A -99.109,B 23.2977,C -0.9908,E1 23.2995,E2 546.2166} C_DIS
LIN {X -17.9954,Y -131.3894,Z 153,A -100.6402,B 23.2977,C -0.9922,E1 23.2953,E2 547.7455} C_DIS
LIN {X -21.0575,Y -130.9335,Z 153,A -101.9808,B 23.2977,C -0.9924,E1 23.2916,E2 549.0868} C_DIS
LIN {X -25.0573,Y -130.225,Z 153,A -103.7816,B 23.2977,C -0.9909,E1 23.2866,E2 550.8934} C_DIS
LIN {X -28.445,Y -129.5279,Z 153,A -105.241,B 23.2976,C -0.9933,E1 23.2826,E2 552.3488} C_DIS
LIN {X -31.8417,Y -128.7366,Z 153,A -106.7495,B 23.2976,C -0.994,E1 23.2785,E2 553.8577} C_DIS
LIN {X -34.9355,Y -127.9316,Z 153,A -108.1327,B 23.2976,C -0.9948,E1 23.2748,E2 555.2412} C_DIS
LIN {X -37.6199,Y -127.1662,Z 153,A -109.3797,B 23.2976,C -0.9937,E1 23.2715,E2 556.4931} C_DIS
LIN {X -41.1185,Y -126.0804,Z 153,A -110.9306,B 23.2975,C -0.9964,E1 23.2673,E2 558.0401} C_DIS
LIN {X -44.2016,Y -125.0328,Z 153,A -112.3432,B 23.2975,C -0.9973,E1 23.2636,E2 559.4533} C_DIS
LIN {X -46.7537,Y -124.0987,Z 153,A -113.5548,B 23.2975,C -0.9967,E1 23.2604,E2 560.6692} C_DIS
LIN {X -50.3438,Y -122.6887,Z 153,A -115.1933,B 23.2973,C -0.9997,E1 23.2562,E2 562.3041} C_DIS
LIN {X -52.9218,Y -121.5965,Z 153,A -116.4161,B 23.2973,C -1.0004,E1 23.253,E2 563.5282} C_DIS
LIN {X -56.2112,Y -120.1124,Z 153,A -117.9642,B 23.2973,C -1.0027,E1 23.2491,E2 565.0745} C_DIS
LIN {X -59.4176,Y -118.5604,Z 153,A -119.5168,B 23.2972,C -1.0039,E1 23.2452,E2 566.6284} C_DIS
LIN {X -62.3953,Y -117.0207,Z 153,A -120.8085,B 23.2968,C -1.0132,E1 23.2421,E2 567.9005} C_DIS
LIN {X -64.6098,Y -115.8127,Z 153,A -122.1833,B 23.2973,C -1.0014,E1 23.2386,E2 569.3095} C_DIS
LIN {X -68.2571,Y -113.7013,Z 153,A -123.9501,B 23.297,C -1.0066,E1 23.2344,E2 571.0689} C_DIS
LIN {X -71.8472,Y -111.4674,Z 153,A -125.779,B 23.297,C -1.0093,E1 23.2301,E2 572.8972} C_DIS
LIN {X -75.2428,Y -109.2035,Z 153,A -127.5911,B 23.297,C -1.0099,E1 23.2259,E2 574.7142} C_DIS
LIN {X -78.8584,Y -106.6225,Z 153,A -129.4261,B 23.2966,C -1.0172,E1 23.2218,E2 576.5378} C_DIS
LIN {X -81.8631,Y -104.3325,Z 153,A -131.1431,B 23.2966,C -1.0162,E1 23.218,E2 578.2639} C_DIS
LIN {X -85.1619,Y -101.6577,Z 153,A -132.9964,B 23.2966,C -1.0189,E1 23.214,E2 580.1182} C_DIS
LIN {X -88.1572,Y -99.0723,Z 153,A -134.75,B 23.2965,C -1.0202,E1 23.2103,E2 581.8758} C_DIS
LIN {X -91.315,Y -96.1695,Z 153,A -136.4882,B 23.2961,C -1.0293,E1 23.2067,E2 583.5987} C_DIS
LIN {X -93.7705,Y -93.7768,Z 153,A -138.0946,B 23.2962,C -1.0268,E1 23.2035,E2 585.2188} C_DIS
LIN {X -96.7553,Y -90.6941,Z 153,A -139.9413,B 23.296,C -1.0312,E1 23.2,E2 587.0629} C_DIS
LIN {X -99.6373,Y -87.5181,Z 153,A -141.7662,B 23.2958,C -1.0367,E1 23.1966,E2 588.8828} C_DIS
LIN {X -102.4123,Y -84.254,Z 153,A -143.5633,B 23.2955,C -1.0435,E1 23.1934,E2 590.6715} C_DIS
LIN {X -104.5525,Y -81.5829,Z 153,A -145.1337,B 23.2955,C -1.0429,E1 23.1906,E2 592.2514} C_DIS
LIN {X -107.0142,Y -78.3253,Z 153,A -146.832,B 23.2952,C -1.0503,E1 23.1878,E2 593.9397} C_DIS
LIN {X -109.2246,Y -75.212,Z 153,A -148.5917,B 23.2952,C -1.0495,E1 23.185,E2 595.7108} C_DIS
LIN {X -111.4589,Y -71.8604,Z 153,A -150.231,B 23.2949,C -1.0586,E1 23.1825,E2 597.336} C_DIS
LIN {X -113.5685,Y -68.4767,Z 153,A -152.0485,B 23.2949,C -1.0589,E1 23.1798,E2 599.1628} C_DIS
LIN {X -115.8106,Y -64.6136,Z 153,A -153.903,B 23.2945,C -1.0675,E1 23.1773,E2 601.0057} C_DIS
LIN {X -117.5582,Y -61.3716,Z 153,A -155.5338,B 23.2944,C -1.0702,E1 23.1751,E2 602.6392} C_DIS
LIN {X -119.1249,Y -58.2732,Z 153,A -157.0398,B 23.2942,C -1.0741,E1 23.1733,E2 604.1439} C_DIS
LIN {X -120.7132,Y -54.9119,Z 153,A -158.6264,B 23.294,C -1.0795,E1 23.1714,E2 605.726} C_DIS
LIN {X -122.0205,Y -51.9411,Z 153,A -160.0245,B 23.2938,C -1.0838,E1 23.1699,E2 607.1217} C_DIS
LIN {X -123.1097,Y -49.2994,Z 153,A -161.3261,B 23.2938,C -1.0845,E1 23.1685,E2 608.4294} C_DIS
LIN {X -124.4725,Y -45.7557,Z 153,A -162.9271,B 23.2935,C -1.091,E1 23.1669,E2 610.0235} C_DIS
LIN {X -125.5642,Y -42.669,Z 153,A -164.3496,B 23.2933,C -1.0949,E1 23.1656,E2 611.4449} C_DIS
LIN {X -126.3947,Y -40.1347,Z 153,A -165.5264,B 23.2932,C -1.0974,E1 23.1646,E2 612.6228} C_DIS
LIN {X -127.4204,Y -36.7518,Z 153,A -167.0245,B 23.2929,C -1.1033,E1 23.1634,E2 614.115} C_DIS
LIN {X -128.2157,Y -33.8703,Z 153,A -168.3403,B 23.2928,C -1.1062,E1 23.1625,E2 615.4318} C_DIS
LIN {X -129.1074,Y -30.3034,Z 153,A -169.9401,B 23.2926,C -1.1106,E1 23.1614,E2 617.0306} C_DIS
LIN {X -129.7937,Y -27.2141,Z 153,A -171.3151,B 23.2924,C -1.1145,E1 23.1606,E2 618.4043} C_DIS
LIN {X -130.402,Y -24.1312,Z 153,A -172.6802,B 23.2922,C -1.1185,E1 23.1599,E2 619.7681} C_DIS
LIN {X -130.9335,Y -21.0575,Z 153,A -174.0354,B 23.292,C -1.1224,E1 23.1593,E2 621.122} C_DIS
LIN {X -131.3827,Y -18.0423,Z 153,A -175.3508,B 23.2918,C -1.1267,E1 23.1587,E2 622.435} C_DIS
LIN {X -131.771,Y -14.9475,Z 153,A -176.7164,B 23.2917,C -1.1302,E1 23.1583,E2 623.8005} C_DIS
LIN {X -132.0796,Y -11.9161,Z 153,A -178.0383,B 23.2915,C -1.1342,E1 23.1579,E2 625.1208} C_DIS
LIN {X -132.3162,Y -8.9114,Z 153,A -179.3444,B 23.2913,C -1.1382,E1 23.1577,E2 626.4252} C_DIS
LIN {X -132.5422,Y -4.4248,Z 153,A 178.7006,B 23.2911,C -1.1439,E1 23.1574,E2 628.3786} C_DIS
LIN {X -132.6079,Y -1.4685,Z 153,A 177.389,B 23.2909,C -1.1465,E1 23.1574,E2 629.692} C_DIS
LIN {X -132.5835,Y 2.9359,Z 153,A 175.3412,B 23.2909,C -1.1463,E1 23.1574,E2 631.7537} C_DIS
LIN {X -132.4459,Y 6.6731,Z 153,A 173.8258,B 23.2905,C -1.156,E1 23.1576,E2 633.2543} C_DIS
LIN {X -132.2373,Y 9.9928,Z 153,A 172.3808,B 23.2903,C -1.1603,E1 23.1579,E2 634.6978} C_DIS
LIN {X -131.935,Y 13.4218,Z 153,A 170.9149,B 23.29,C -1.166,E1 23.1583,E2 636.1585} C_DIS
LIN {X -131.5903,Y 16.4617,Z 153,A 169.5812,B 23.2898,C -1.1698,E1 23.1587,E2 637.4913} C_DIS
LIN {X -131.2511,Y 18.9631,Z 153,A 168.4202,B 23.2898,C -1.1703,E1 23.1592,E2 638.6586} C_DIS
LIN {X -130.6787,Y 22.5851,Z 153,A 166.8815,B 23.2895,C -1.1774,E1 23.1599,E2 640.1892} C_DIS
LIN {X -130.1091,Y 25.6637,Z 153,A 165.516,B 23.2893,C -1.1812,E1 23.1606,E2 641.5537} C_DIS
LIN {X -129.4621,Y 28.7502,Z 153,A 164.142,B 23.2891,C -1.185,E1 23.1614,E2 642.9267} C_DIS
LIN {X -128.8593,Y 31.3326,Z 153,A 162.9564,B 23.2891,C -1.187,E1 23.1622,E2 644.1149} C_DIS
LIN {X -127.9316,Y 34.9355,Z 153,A 161.3646,B 23.2887,C -1.1927,E1 23.1633,E2 645.7019} C_DIS
LIN {X -127.0465,Y 38.0288,Z 153,A 159.9625,B 23.2886,C -1.1966,E1 23.1644,E2 647.103} C_DIS
LIN {X -126.0804,Y 41.1185,Z 153,A 158.5521,B 23.2884,C -1.2005,E1 23.1656,E2 648.5123} C_DIS
LIN {X -125.2255,Y 43.6458,Z 153,A 157.3806,B 23.2882,C -1.2033,E1 23.1666,E2 649.6838} C_DIS
LIN {X -124.065,Y 46.8437,Z 153,A 155.8981,B 23.288,C -1.2073,E1 23.1681,E2 651.1652} C_DIS
LIN {X -122.6887,Y 50.3438,Z 153,A 154.2694,B 23.2878,C -1.2121,E1 23.1698,E2 652.7915} C_DIS
LIN {X -121.6107,Y 52.8889,Z 153,A 153.0598,B 23.2877,C -1.2151,E1 23.1711,E2 654.0007} C_DIS
Enddeposition()
END
